# B&R Automation Studio project NAEUL004C00R13L518F00 (part 70)

#### Local.var - Do Not Change!!!
```iecst
(*2019-04-16*)
(**)
(*Local Action, State & Status*)
VAR
	eStatus : eFBStatus := Idle;
	udiStatus : UDINT := 0;
END_VAR
(**)
(*Local Alarm*)
VAR
	tyAlmData : tyAlmDat;
	a_tyAlmText : ARRAY[10000..10099] OF tyAlmTxt := [(sAlmText:='Magazine Not Present While Pushing Board Into Magazine',sRcyText:='Insert Magazine To Continue Operation.'),(sAlmText:='Conveyor Outlet Sensor Timeout Alarm',sRcyText:='Check Conveyor Outlet Sensor'),(sAlmText:='Conveyor Inlet Sensor Timeout Alarm',sRcyText:='Check Conveyor Inlet Sensor'),(sAlmText:='Clear Sensor Activated When Board Transfer In',sRcyText:='Please Check The Sensitivity of Pusher Conveyor Outlet Sensor'),(sAlmText:='Magazine Width Check Timeout Alarm',sRcyText:='Magazine Is Not Set In Correct Width'),(sAlmText:='Pusher AntiJam Sensor On',sRcyText:='Board Jam During Pusher Is Extending'),(sAlmText:='No Barcode Detected.',sRcyText:='Check The Barcode Position.'),(sAlmText:='Return Code Feedback Time Out.',sRcyText:='Reset And Resume Operation.'),(sAlmText:='Board Lost Before Traversing.',sRcyText:='Check If Outlet sensor False Triggerred or Board Stuck in Middle '),(sAlmText:='Inlet and outlet same time sensing error.',sRcyText:='Please Ensure No Blockage At Inlet Sensor.'),(sAlmText:='OpCon Error',sRcyText:='OpCon Error'),(sAlmText:='ScanningTime Out Error',sRcyText:='Ensure Connection for Scan Completed Signal'),(sAlmText:='Anti Crash Sensor Activated Before Traversing',sRcyText:='Please Check Board is away from Clear Sensor'),87((0))];
END_VAR
(**)
(*Local Output*)
VAR
	sStepTxt : STRING[80];
	bPaused : BOOL;
END_VAR
(**)
VAR
	eUSSMEMAAct1 : eSMEMAAction;
	eUSSMEMAAct2 : eSMEMAAction;
	eUSSMEMAAct3 : eSMEMAAction;
	eDSSMEMAAct1 : eSMEMAAction;
	eDSSMEMAAct2 : eSMEMAAction;
	eDSSMEMAAct3 : eSMEMAAction;
	eConvAct : eConvAction;
	eAWAct : eAWAction;
	eAWPushOrPullerAct : eAWAction;
	eTravAct : eTravAction;
	eLifAct : eLifterAction;
	eInletPneuAct : ePneuAction;
	eOutletPneuAct : ePneuAction;
	eOutletPneuAct2 : ePneuAction;
	eOutletPneuAct3 : ePneuAction;
	eStopperAct1 : ePneuAction;
	eStopperAct2 : ePneuAction;
	eStopperAct3 : ePneuAction;
	udiJogSpeed : UDINT := 290000;
END_VAR
(**)
VAR
	eTravLifPosGo : eTravLifULPos;
	a_bMagDis : ARRAY[1..3] OF BOOL;
	a_bMagRej : ARRAY[1..3] OF BOOL;
	bInitConv : BOOL;
	bOpsInitDone : BOOL;
	bUSComm : BOOL;
	bEntBrd : BOOL;
	bDSComm : BOOL;
	bExitBrd : BOOL;
	bTravLifMove : BOOL;
	bUSWidthChkBrdExist : BOOL := TRUE;
	bStopperExtStep : BOOL;
	fbWaitTimer : TON := (PT:=T#2s);
	fbWidthChkSenOnTim : TON := (PT:=T#5s);
	fbWidthChkSenOffTim : TON := (PT:=T#1s);
END_VAR
(*Step Logger*)
VAR
	bClsLog : BOOL;
	blog : BOOL;
	logStep : ARRAY[0..999] OF eTravLifULStep;
	logIndexStep : INT;
	eGotoOpsStepDummy : eTravLifULStep;
END_VAR
(**)
(*Local Input*)
VAR
	udiRstErr : UDINT := 0;
	bEn : BOOL := TRUE;
	bDis : BOOL := FALSE;
	bRun : BOOL;
	bStop : BOOL;
	bStep : BOOL;
	eULMode : eULMod;
	eULMagazine : eULMag;
	bNonBffrMod : BOOL;
	bBypsGdBadBrd : BOOL;
	bUSAllow : BOOL := TRUE;
	bDSAllow : BOOL := TRUE;
	eUSCommMod1 : eMcSetCommMod;
	eUSCommMod2 : eMcSetCommMod;
	eUSCommMod3 : eMcSetCommMod;
	eDSCommMod1 : eMcSetCommMod;
	eDSCommMod2 : eMcSetCommMod;
	eDSCommMod3 : eMcSetCommMod;
	eUSSMEMAStat1 : eSMEMAAction;
	eUSSMEMAStatus1 : eFBStatus;
	bUSSMEMAUSRdy1 : BOOL;
	bUSSMEMAGdBrdRdy1 : BOOL;
	bUSSMEMATransporting1 : BOOL;
	bUSSMEMAConvStart1 : BOOL;
	bUSSMEMAConvStop1 : BOOL;
	eUSSMEMAStat2 : eSMEMAAction;
	eUSSMEMAStatus2 : eFBStatus;
	bUSSMEMAUSRdy2 : BOOL;
	bUSSMEMAGdBrdRdy2 : BOOL;
	bUSSMEMATransporting2 : BOOL;
	bUSSMEMAConvStart2 : BOOL;
	bUSSMEMAConvStop2 : BOOL;
	eUSSMEMAStat3 : eSMEMAAction;
	eUSSMEMAStatus3 : eFBStatus;
	bUSSMEMAUSRdy3 : BOOL;
	bUSSMEMAGdBrdRdy3 : BOOL;
	bUSSMEMATransporting3 : BOOL;
	bUSSMEMAConvStart3 : BOOL;
	bUSSMEMAConvStop3 : BOOL;
	eDSSMEMAStat1 : eSMEMAAction;
	eDSSMEMAStatus1 : eFBStatus;
	bDSSMEMADSRdy1 : BOOL;
	bDSSMEMAConvStart1 : BOOL;
	eDSSMEMAStat2 : eSMEMAAction;
	eDSSMEMAStatus2 : eFBStatus;
	bDSSMEMADSRdy2 : BOOL;
	bDSSMEMAConvStart2 : BOOL;
	eDSSMEMAStat3 : eSMEMAAction;
	eDSSMEMAStatus3 : eFBStatus;
	bDSSMEMADSRdy3 : BOOL;
	bDSSMEMAConvStart3 : BOOL;
	bUSHermesUSRdy1 : BOOL;
	bUSHermesUSGdRdy1 : BOOL;
	bUSHermesTransporting1 : BOOL;
	bUSHermesStopTransport1 : BOOL;
	bUSHermesUSRdy2 : BOOL;
	bUSHermesUSGdRdy2 : BOOL;
	bUSHermesTransporting2 : BOOL;
	bUSHermesStopTransport2 : BOOL;
	bUSHermesUSRdy3 : BOOL;
	bUSHermesUSGdRdy3 : BOOL;
	bUSHermesTransporting3 : BOOL;
	bUSHermesStopTransport3 : BOOL;
	bDSHermesDSRdy1 : BOOL;
	bDSHermesTransporting1 : BOOL;
	bDSHermesStopTransport1 : BOOL;
	bDSHermesDSRdy2 : BOOL;
	bDSHermesTransporting2 : BOOL;
	bDSHermesStopTransport2 : BOOL;
	bDSHermesDSRdy3 : BOOL;
	bDSHermesTransporting3 : BOOL;
	bDSHermesStopTransport3 : BOOL;
	eConvStat : eConvAction;
	eConvStatus : eFBStatus;
	eConvDirection : eConvDir;
	bConvHvBrd : BOOL;
	bConvGdBrd : BOOL;
	eAWStat : eAWAction;
	eAWStatus : eFBStatus;
	bAWWidthPosDiff : BOOL;
	eTravStat : eTravAction;
	eTravStatus : eFBStatus;
	eLifStat : eLifterAction;
	eLifStatus : eFBStatus;
	eInletPneuStat : ePneuAction;
	eInletPneuStatus : eFBStatus;
	bInletPneuCls : BOOL;
	eOutletPneuStat : ePneuAction;
	eOutletPneuStatus : eFBStatus;
	bConvLftSen : BOOL;
	bConvRgtSen : BOOL;
	bMagTransferBrd1 : BOOL;
	bMagTransferBrd2 : BOOL;
	bMagTransferBrd3 : BOOL;
	bBufferMagPresent1 : BOOL;
	bBufferMagPresent2 : BOOL;
	bBufferMagPresent3 : BOOL;
	sProgNm : STRING[15] := 'Ops TravLifUL';
	bNtSettingsLoadDone : BOOL := TRUE;
	tShutterWaitTmr : TIME := T#0s;
	eMagBuffferActLoad : eLifMagULUpdateData;
	bScanEn : BOOL := FALSE;
	eTCPTopStat : eTCPAction1;
	eTCPTopStatus : eFBStatus;
	sTopMsgRd : STRING[80] := '';
	eTCPBtmStat : eTCPAction1;
	eTCPBtmStatus : eFBStatus;
	sBtmMsgRd : STRING[80] := '';
	bInitInletPneu : BOOL := FALSE;
	bWidthChkErrCmdUnclmp1 : BOOL;
	bWidthChkErrCmdUnclmp2 : BOOL;
	bWidthChkErrCmdUnclmp3 : BOOL;
	bCmdUnclmpFlag : BOOL;
	bPneuUnclmpFBDone : BOOL;
END_VAR
(**)
(*Local*)
VAR
	bRstErr : BOOL;
	udiRstErrOld : UDINT;
	bInitDone : BOOL;
	bInitialDone : BOOL;
	eOpsStep : eTravLifULStep := TravLifULStepNA;
	eGotoOpsStep : eTravLifULStep := TravLifULStepInitConv;
	tyParamTravLif : tyParamTravLifUL;
	bOpsModGonethrough : BOOL;
	udiMagPresentTm1 : UDINT;
	udiMagPresentTm : UDINT;
	udiCmpTm : UDINT;
	udiCount : UDINT;
	udi : UDINT;
	bGdChk : BOOL;
	udiPosAllwGo : UDINT;
	a_bPosAllwSigOn : ARRAY[1..3] OF BOOL;
	a_udiPosAllwSum : ARRAY[1..3] OF UDINT;
	a_tyMagAllwBffrStat : ARRAY[1..3] OF tyBffrStat;
	a_udiMagAllwMagPresentTm : ARRAY[1..3] OF UDINT;
	a_udiMagAllwPriority : ARRAY[1..3] OF UDINT;
	bBrdOnSen : BOOL;
	bBrdOnStopperSen : BOOL;
	bStopperBrdOnSen : BOOL;
	bConvInSenOn : BOOL;
	bConvOutSenOn : BOOL;
	bLocalUSRdy1 : BOOL;
	bLocalUSGdRdy1 : BOOL;
	bLocalUSRdy2 : BOOL;
	bLocalUSGdRdy2 : BOOL;
	bLocalUSRdy3 : BOOL;
	bLocalUSGdRdy3 : BOOL;
	bLocalDSRdy1 : BOOL;
	bLocalDSRdy2 : BOOL;
	bLocalDSRdy3 : BOOL;
	bSkipCloseInletShutter : BOOL;
	tConvRgtSenOff : TON := (PT:=T#100ms);
	tConvLftSenOff : TON := (PT:=T#100ms);
	tEntBoardTimoutErr : TON := (PT:=T#6s);
	tExitBoardTimoutErr : TON := (PT:=T#10s);
	tTravLiftInPos : TON := (PT:=T#100ms);
	bTravLifInDSPos : BOOL;
	bSelfTest : BOOL;
	bLifterBtmPosDiff : BOOL;
	bLifterAPosDiff : BOOL;
	bLifterBPosDiff : BOOL;
	bBypCurtainSenPB : BOOL;
	bBypCurtainSenCtrl : BOOL;
	bBypCurtainSensorPBLED : BOOL;
	bMagWidthChkDis : BOOL;
	fbRstCurtain : TON := (PT:=T#1m);
	fb2SenTm : TON;
	p_eStopperAct : REFERENCE TO ePneuAction;
	p_eStopperStat : REFERENCE TO ePneuAction;
	p_eStopperStatus : REFERENCE TO eFBStatus;
	p_bStopperBlk : REFERENCE TO BOOL;
	p_eLocalUSCommMod : REFERENCE TO eMcSetCommMod;
	p_eLocalDSCommMod : REFERENCE TO eMcSetCommMod;
	p_bLocalUSRdy : REFERENCE TO BOOL;
	p_bLocalUSGdRdy : REFERENCE TO BOOL;
	p_bLocalDSRdy : REFERENCE TO BOOL;
	p_eLocalUSSMEMAAct : REFERENCE TO eSMEMAAction;
	p_eLocalUSSMEMAStat : REFERENCE TO eSMEMAAction;
	p_eLocalUSSMEMAStatus : REFERENCE TO eFBStatus;
	p_bLocalUSSMEMAUSRdy : REFERENCE TO BOOL;
	p_bLocalUSSMEMAGdBrdRdy : REFERENCE TO BOOL;
	p_bLocalUSSMEMATransporting : REFERENCE TO BOOL;
	p_bLocalUSSMEMAConvStart : REFERENCE TO BOOL;
	p_bLocalUSSMEMAConvStop : REFERENCE TO BOOL;
	p_eLocalDSSMEMAAct : REFERENCE TO eSMEMAAction;
	p_eLocalDSSMEMAStat : REFERENCE TO eSMEMAAction;
	p_eLocalDSSMEMAStatus : REFERENCE TO eFBStatus;
	p_bLocalDSSMEMADSRdy : REFERENCE TO BOOL;
	p_bLocalDSSMEMAConvStart : REFERENCE TO BOOL;
	p_bLocalUSHermesUSRdy : REFERENCE TO BOOL;
	p_bLocalUSHermesUSGdRdy : REFERENCE TO BOOL;
	p_bLocalUSHermesTransporting : REFERENCE TO BOOL;
	p_bLocalUSHermesStopTransport : REFERENCE TO BOOL;
	p_bLocalDSHermesDSRdy : REFERENCE TO BOOL;
	p_bLocalDSHermesTransporting : REFERENCE TO BOOL;
	p_bLocalDSHermesStopTransport : REFERENCE TO BOOL;
	fbBypCurtainPBLEDBlinkTm : TON := (IN:=FALSE,PT:=T#500ms,Q:=FALSE,ET:=0,StartTime:=0,M:=FALSE,Restart:=0);
	eLocalUSCommMod : eMcSetCommMod;
	bWait : BOOL;
END_VAR
(*Inlet stopper*)
VAR
	eInletStopperAct : ePneuAction;
END_VAR
(*Scanner Param *)
VAR
	eTCPTopAct : eTCPAction1;
	eTCPBtmAct : eTCPAction1;
	sBarcode : STRING[80];
	bPass : BOOL;
END_VAR
(*xml*)
VAR
	tyOpConParam : tyLocationParam;
	tyOpConMsgReq : eOpConMsgType;
	bJamStarted : BOOL := FALSE;
	bWaitMagChkRetCode : BOOL;
	fbIdleTm : TON := (PT:=T#3m);
	fbReturnCodeTO : TON := (PT:=T#30s);
END_VAR
(**)
VAR
	tyPartReceive : tyOpConPartReceive;
	tyPartProcessedItems : tyOpConPartProcessed; (*Output*)
	tyMagCoordinate : tyMagCoord;
	diTemp : DINT;
	bHermesBC : BOOL;
	diMagBrdQty : ARRAY[1..3] OF DINT;
	bPLCGrabPic : BOOL;
	asMagEntered : ARRAY[0..4] OF STRING[10];
	udiModuleNum : UDINT := 6621;
END_VAR
(*Siemen *)
VAR
	bAllwExitMag1 : BOOL;
	bAllwExitMag2 : BOOL;
	bAllwExitMag3 : BOOL;
	fbInletStopperOffTim : TON := (PT:=T#1s);
END_VAR
(*Bosch Scanner*)
VAR
	bScannerEn : BOOL;
	bTCPScanner : BOOL;
	bSignalTrigMagOutEn : BOOL;
	bTCPScannerEn : BOOL;
	fbScanTimOut : TON := (PT:=T#10s);
	bStartScanSig : BOOL;
	bPCBExitMag1 : BOOL;
	bPCBExitMag2 : BOOL;
	bPCBExitMag3 : BOOL;
	usiScanCntr : USINT;
END_VAR
```

### OpsMagConvUL.typ - Do Not Change!!!
```iecst
(*2018-12-11*)
(**)
(*Sequence*)

TYPE
	eMagConvULStep :
		(
		MagConvULStepNA,
		MagConvULStepInitMag,
		MagConvULStepSafetyBarExtCtrl,
		MagConvULStepMagUSComm,
		MagConvULStepInitAWPneu,
		MagConvULStepInitMagEnt,
		MagConvULStepInitMagFixClp,
		MagConvULStepInitMagConv,
		MagConvULStepMagEnt,
		MagConvULStepMagEntMnl,
		MagConvULStepSelClampCtrl,
		MagConvULStepVerifyMag,
		MagConvULStepChkMag,
		MagConvULStepSafetyBarExt,
		MagConvULStepSafetyBarRet,
		MagConvULStepMagAWEngage,
		MagConvULStepMagAWDisengage,
		MagConvULStepMagAWHm,
		MagConvULStepMagAWMov,
		MagConvULStepMagEntMESStdByChk,
		MagConvULStepBffrStatChk,
		MagConvULStepMagCmp,
		MagConvULStepMtyBffr,
		MagConvULStepNxtLoadBffr,
		MagConvULStepBffrUSComm,
		MagConvULStepBffrEntBrd,
		MagConvULStepUpdateBffr,
		MagConvULStepLoadBffr,
		MagConvULStepMagExtMESStdByChk,
		MagConvULStepMagExitClampCtrl,
		MagConvULStepMagExitSafeBarCtrl,
		MagConvULStepMagFullDSComm,
		MagConvULStepMagFullExit,
		MagConvULStepMagExitMnl,
		MagConvULStepMagHalfExitMnl,
		MagConvULStepMagExitedWait,
		MagConvULStepMagExitedAGVWait
		);
	eLifMagULUpdateData :
		(
		BufferActLoadWhenStarted,
		BufferActLoadWhenCompleted
		);
END_TYPE
```

### OpsMagConvUL1.var - Change By Project
```iecst
(*2019-03-25*)
(**)
(*Action & State & Status*)
(**)
(*Alarm*)
VAR
	p_OpsMagConvUL1AlmData : UDINT;
	p_OpsMagConvUL1AlmData1 : UDINT;
END_VAR
(**)
(*Output*)
VAR
	p_OpsMagConvUL1StepTxt : UDINT;
	p_OpsMagConvUL1Paused : UDINT;
END_VAR
(**)
VAR
	p_OpsMagConvUL1BufferAct : UDINT;
	p_OpsMagConvUL1MagConv2ClpAct : UDINT;
	p_OpsMagConvUL1USSMEMAAct : UDINT;
	p_OpsMagConvUL1AGVMagAct : UDINT;
	p_OpsMagConvUL1MagFullExit : UDINT;
	p_OpsMagConvUL1IncorrectMagModel : UDINT;
	p_OpsMagConvUL1MagSizeL : UDINT;
END_VAR
(**)
VAR
	p_OpsMagConvUL1InitDone : UDINT;
	p_OpsMagConvUL1MagBffrAvl : UDINT;
	p_OpsMagConvUL1NewMagAllw : UDINT;
	p_OpsMagConvUL1RlsMagAllw : UDINT;
	p_OpsMagConvUL1EjectMESStep : UDINT;
	p_OpsMagConvUL1EjectMagNotAllw : UDINT;
	p_OpsMagConvUL1StepSelClampCtrl : UDINT;
	p_OpsMagConvUL1StepMagExitedWait : UDINT;
	p_OpsMagConvUL1NewMagVerified : UDINT;
	p_OpsMagConvUL1StepUSCom : UDINT;
	p_OpsMagConvUL1StepBffrLoad : UDINT;
	p_OpsMagConvUL1StepPLCGrab : UDINT;
END_VAR
(**)
VAR
	p_OpsMagConvUL1SafetyBarAct : UDINT;
	p_OpsMagConvUL1MagAWEngageAct : UDINT;
	p_OpsMagConvUL1MagAWAct : UDINT;
	p_OpsAGVCommRdy1 : UDINT;
END_VAR
(**)
VAR
	p_OpsMagConvUL1USSOTAct : UDINT;
	p_OpsMagConvUL1DSSOTAct : UDINT;
	p_OpsMagConvUL1MsgReq : UDINT;
	p_OpsMagConvUL1UnclmpDone : UDINT;
	p_OpsMagConvUL1MagAllwGo : UDINT;
	p_OpsMagConvUL1ReadRFID : UDINT;
	p_OpsMagConvUL1WriteRFID : UDINT;
	p_OpsMagConvUL1AWDone : UDINT;
	p_OpsMagConvUL1SlotUpdtDone : UDINT;
	p_OpsMagConvUL1AcptTm : UDINT;
	p_OpsMagConvUL1MESAcptCond : UDINT;
	p_OpsMagConvUL1MagExitedWait : UDINT;
	p_OpsMagConvUL1TLMuteBuzz : UDINT;
	p_OpsMagConvUL1MagFullInfo : UDINT;
END_VAR
(**)
```

### Program Logical/Operations/MagConv_StationaryPlat/OpsMagConvUL1 (IEC) - 1.00.0 - 

#### InputRef.var
```iecst
(*2019-04-16*)
(**)
(*General*)
VAR
	p_udiRstErr : REFERENCE TO UDINT;
	p_bEn : REFERENCE TO BOOL;
	p_bDis : REFERENCE TO BOOL;
	p_bRun : REFERENCE TO BOOL;
	p_bStop : REFERENCE TO BOOL;
	p_bStep : REFERENCE TO BOOL;
END_VAR
(**)
(*Configuration*)
VAR
	p_sProgNm : REFERENCE TO STRING[15];
	p_bNtSettingsLoadDone : REFERENCE TO BOOL;
END_VAR
(**)
VAR
	p_usiMagConv : REFERENCE TO USINT;
	p_bInfoEn : REFERENCE TO BOOL;
END_VAR
(**)
VAR
	pa_bMagDis : REFERENCE TO ARRAY[1..3] OF BOOL;
	pa_bMagRej : REFERENCE TO ARRAY[1..3] OF BOOL;
	pa_bMagChangeOverBlk : REFERENCE TO ARRAY[1..4] OF BOOL;
	p_bMagPropDiffBlk : REFERENCE TO BOOL;
	p_bUSAllow : REFERENCE TO BOOL;
	p_bAllwChgWidth : REFERENCE TO BOOL;
	p_bAllwChgSlot : REFERENCE TO BOOL;
	p_bChgMagWidth : REFERENCE TO BOOL;
	p_bChgMagSlot : REFERENCE TO BOOL;
	p_bMagOrientChkSenPrep : REFERENCE TO BOOL;
	p_bDIMagFixedClampSen : REFERENCE TO BOOL;
	p_eCustomerReq : REFERENCE TO eCustomer;
END_VAR
(*Siemen MES*)
VAR
	p_tyResponseFromMES : REFERENCE TO tyStatPlatformFromMES;
	p_bOpsTravLifAllwExitMag : REFERENCE TO BOOL;
	p_diMcParamMESResponseTO : REFERENCE TO DINT;
	p_bMcParamMESEn : REFERENCE TO BOOL;
	p_bAutoRcpForceExitMag : REFERENCE TO BOOL;
	p_dtCurrDT : REFERENCE TO DATE_AND_TIME;
	p_dtOpsMagConvUL1AcptTm : REFERENCE TO DATE_AND_TIME;
	p_dtOpsMagConvUL2AcptTm : REFERENCE TO DATE_AND_TIME;
	p_dtOpsMagConvUL3AcptTm : REFERENCE TO DATE_AND_TIME;
	p_iOpsMagConvUL1MESAcptCond : REFERENCE TO INT;
	p_iOpsMagConvUL2MESAcptCond : REFERENCE TO INT;
	p_iOpsMagConvUL3MESAcptCond : REFERENCE TO INT;
	p_bOpsMagConvUL2MagExitedWait : REFERENCE TO BOOL;
	p_bOpsMagConvUL3MagExitedWait : REFERENCE TO BOOL;
	p_usiUIHcomModchanged : REFERENCE TO USINT;
	p_bNtParamAutoRcpF1ArbitraryType : REFERENCE TO BOOL;
END_VAR
(**)
VAR
	p_bNewMag : REFERENCE TO BOOL;
	p_bRlsMag : REFERENCE TO BOOL;
END_VAR
(**)
VAR
	p_bConvInitDone : REFERENCE TO BOOL;
	p_bConvHvBrd : REFERENCE TO BOOL;
	p_bConvGdBrd : REFERENCE TO BOOL;
END_VAR
(**)
VAR
	p_tyBufferStat1 : REFERENCE TO tyBffrStat;
	p_tyBufferStat2 : REFERENCE TO tyBffrStat;
	p_tyBufferStat3 : REFERENCE TO tyBffrStat;
END_VAR
(**)
VAR
	p_bMagClampRS1 : REFERENCE TO BOOL;
	p_bMagClampRS2 : REFERENCE TO BOOL;
	p_bMagClampRS3 : REFERENCE TO BOOL;
END_VAR
(**)
VAR
	p_bMagEntrySen : REFERENCE TO BOOL;
	p_bMagEntrySen1 : REFERENCE TO BOOL;
	p_bMagEntrySen2 : REFERENCE TO BOOL;
	p_bMagEntrySen3 : REFERENCE TO BOOL;
END_VAR
(**)
VAR
	p_bMagPresentSen : REFERENCE TO BOOL;
	p_bMagPresentSen1 : REFERENCE TO BOOL;
	p_bMagPresentSen2 : REFERENCE TO BOOL;
	p_bMagPresentSen3 : REFERENCE TO BOOL;
END_VAR
(**)
VAR
	p_bBufferMagPresent1 : REFERENCE TO BOOL;
	p_bBufferMagPresent2 : REFERENCE TO BOOL;
	p_bBufferMagPresent3 : REFERENCE TO BOOL;
END_VAR
(**)
VAR
	p_bBufferMagRemoved : REFERENCE TO BOOL;
	p_bBufferMagRemoved1 : REFERENCE TO BOOL;
	p_bBufferMagRemoved2 : REFERENCE TO BOOL;
	p_bBufferMagRemoved3 : REFERENCE TO BOOL;
END_VAR
(**)
VAR
	p_dtBufferMagPresentTm1 : REFERENCE TO DATE_AND_TIME;
	p_dtBufferMagPresentTm2 : REFERENCE TO DATE_AND_TIME;
	p_dtBufferMagPresentTm3 : REFERENCE TO DATE_AND_TIME;
END_VAR
(**)
VAR
	p_eBufferStat : REFERENCE TO eBufferAction;
	p_eBufferStatus : REFERENCE TO eFBStatus;
END_VAR
(**)
VAR
	p_eMagConv2ClpStat : REFERENCE TO eMagConv2ClpAction;
	p_eMagConv2ClpStatus : REFERENCE TO eFBStatus;
	p_bMagConv2ClpHvMag : REFERENCE TO BOOL;
END_VAR
(**)
VAR
	p_eUSSMEMAStat : REFERENCE TO eSMEMAAction;
	p_eUSSMEMAStatus : REFERENCE TO eFBStatus;
	p_bUSSMEMATransporting : REFERENCE TO BOOL;
	p_bUSSMEMAConvStart : REFERENCE TO BOOL;
	p_bUSSMEMAConvStop : REFERENCE TO BOOL;
END_VAR
(**)
VAR
	p_eAGVMagStat : REFERENCE TO eAGVMagAction;
	p_eAGVMagStatus : REFERENCE TO eFBStatus;
	p_bAGVMagMcRunRdy : REFERENCE TO BOOL;
	p_tyAGVToDTMag : REFERENCE TO tyTagAGVToDTMag;
END_VAR
(**)
VAR
	p_eSelClampCtrlStat : REFERENCE TO ePneuAction;
	p_eSelClampCtrlStatus : REFERENCE TO eFBStatus;
END_VAR
(**)
VAR
	p_bOutShutterExtended : REFERENCE TO BOOL;
END_VAR
(**)
VAR
	p_bDIMagConvHeightSen : REFERENCE TO BOOL;
	p_bDIMagConvSelUnclampRS : REFERENCE TO BOOL;
	p_bDIMagConvCAB717Sen : REFERENCE TO BOOL;
	p_bDIMagConvSmallSen : REFERENCE TO BOOL;
	p_bDIMagConvLargeSen : REFERENCE TO BOOL;
	p_bDIOutShutterClosedRS : REFERENCE TO BOOL;
END_VAR
(**)
VAR
	p_eSafetyBarStat : REFERENCE TO ePneuAction;
	p_eSafetyBarStatus : REFERENCE TO eFBStatus;
	p_bSafetyBarExtended : REFERENCE TO BOOL;
	p_bSafetyBarRetracted : REFERENCE TO BOOL;
END_VAR
(**)
VAR
	p_eMagAWEngageStat : REFERENCE TO ePneuAction;
	p_eMagAWEngageStatus : REFERENCE TO eFBStatus;
	p_eConvStat : REFERENCE TO eConvAction;
	p_eConvStatus : REFERENCE TO eFBStatus;
END_VAR
(**)
VAR
	p_eMagAWStat : REFERENCE TO eMagAWAction;
	p_eMagAWStatus : REFERENCE TO eFBStatus;
	p_bMagAWEngaging : REFERENCE TO BOOL;
	p_bMagAWErr : REFERENCE TO BOOL;
	p_bMagAWOpenLimit : REFERENCE TO BOOL;
	p_bMagAWCloseLimit : REFERENCE TO BOOL;
END_VAR
(**)
VAR
	p_eUSSOTStat : REFERENCE TO eSOTAction;
	p_eUSSOTStatus : REFERENCE TO eFBStatus;
	p_bUSSOTTransporting : REFERENCE TO BOOL;
	p_bUSSOTConvStart : REFERENCE TO BOOL;
	p_bUSSOTConvStop : REFERENCE TO BOOL;
	p_bUSSOTUSRdy : REFERENCE TO BOOL;
	p_bUSSOTUSLargeMagRdy : REFERENCE TO BOOL;
END_VAR
(**)
VAR
	p_eDSSOTStat : REFERENCE TO eSOTAction;
	p_eDSSOTStatus : REFERENCE TO eFBStatus;
	p_bDSSOTConvStart : REFERENCE TO BOOL;
	p_bDSSOTConvStop : REFERENCE TO BOOL;
END_VAR
(**)
VAR
	p_bOpsTravLifExitBrd : REFERENCE TO BOOL;
	p_bOpsTravLifMov : REFERENCE TO BOOL;
END_VAR
(**)
(*Self Test Var*)
VAR
	p_bSelfTest : REFERENCE TO BOOL;
	p_bMcParamMagAWDis : REFERENCE TO BOOL;
	p_bDISOTRcv : REFERENCE TO BOOL;
	p_bDISOTAGVReady : REFERENCE TO BOOL;
END_VAR
(**)
VAR
	p_diProdRcpCurrRcp1Width : REFERENCE TO DINT;
	p_diProdRcpCurrRcp2Width : REFERENCE TO DINT;
	p_sProdRcpCurrRcp1Name : REFERENCE TO STRING[80];
	p_sProdRcpCurrRcp2Name : REFERENCE TO STRING[80];
	p_sMagRcpName : REFERENCE TO DINT;
	p_bOpsTravLifErrCmdUnclmp : REFERENCE TO BOOL;
END_VAR
(**)
VAR
	p_bNtParamAutoRcpPrep : REFERENCE TO BOOL;
	p_bMcParamAutoRcpDis : REFERENCE TO BOOL;
END_VAR
```

#### InputRef_Link.var
```iecst
(*2018-12-11*)
(**)
VAR
	p_bLinkDIMagPresentSen1 : REFERENCE TO BOOL;
	p_bLinkMagConv2Clp1MtrIn : REFERENCE TO BOOL;
	p_bLinkMagConv2Clp1MtrOut : REFERENCE TO BOOL;
	p_bLinkDIMagPresentSen2 : REFERENCE TO BOOL;
	p_bLinkMagConv2Clp2MtrIn : REFERENCE TO BOOL;
	p_bLinkMagConv2Clp2MtrOut : REFERENCE TO BOOL;
	p_bLinkDIMagPresentSen3 : REFERENCE TO BOOL;
	p_bLinkMagConv2Clp3MtrIn : REFERENCE TO BOOL;
	p_bLinkMagConv2Clp3MtrOut : REFERENCE TO BOOL;
	p_bLinkFixedMagClampRS1 : REFERENCE TO BOOL;
	p_bLinkRmtMagClampRS1 : REFERENCE TO BOOL;
	p_bLinkFixedMagClampRS2 : REFERENCE TO BOOL;
	p_bLinkRmtMagClampRS2 : REFERENCE TO BOOL;
	p_bLinkFixedMagClampRS3 : REFERENCE TO BOOL;
	p_bLinkRmtMagClampRS3 : REFERENCE TO BOOL;
	p_bLinkMcParamMagAutoDetTm : REFERENCE TO DINT;
	p_bLinkDIMagEntrySen : REFERENCE TO BOOL;
	p_bLinkNtParamMagModelAutoVerify : REFERENCE TO BOOL;
	p_bLinkMagRcpCurrRcpMagModel : REFERENCE TO USINT;
	p_bLinkNewMagVerified2 : REFERENCE TO BOOL;
	p_bLinkNewMagVerified3 : REFERENCE TO BOOL;
	p_eNtParamProjMagBuffferActLoad : REFERENCE TO eLifMagULUpdateData;
	p_eLinkMcParamMagExMode : REFERENCE TO eMcMagExchangeMode;
END_VAR
(**)
VAR
	p_bMag1OrientationChkSen1 : REFERENCE TO BOOL;
	p_bMagHeightDetSen1 : REFERENCE TO BOOL;
	p_bMagHeightDetEn : REFERENCE TO BOOL;
	p_bMagHeightDetPrep : REFERENCE TO BOOL;
	p_bProjLifTravMnlLoad : REFERENCE TO BOOL;
END_VAR
```

#### Local.var
```iecst
(*2019-04-16*)
(**)
(*Local Action, State & Status*)
VAR
	eStatus : eFBStatus := Idle;
	udiStatus : UDINT := 0;
	udiStatus1 : UDINT := 0;
END_VAR
(**)
(*Local Alarm*)
VAR
	tyAlmData : tyAlmDat;
	tyAlmData1 : tyAlmDat;
	a_tyAlmText : ARRAY[10000..10099] OF tyAlmTxt := [(sAlmText:='Magazine Not Present'),(sAlmText:='Magazine 1 Is Full'),(sAlmText:='Magazine 2 Is Full'),(sAlmText:='Magazine 3 Is Full'),(sAlmText:='Please Insert Good Magazine'),(sAlmText:='Please Insert Bad Magazine'),(sAlmText:='Wrong Magazine Width On Position 1'),(sAlmText:='Wrong Magazine Height On Position 1'),(sAlmText:='Waiting for Unload Magazine 1'),(sAlmText:='Rack/Magazine Auto Width Change Error',sRcyText:='Rack/Magazine Auto Width Motor Error While Doing Width Change'),(sAlmText:='Magazine 1 Auto Width Limit Sensor Activated, Ensure Senor Is Cleared Or Magazine Is Empty ',sRcyText:='Please make sure magazine wall is clear from limit sensor and there is no object in the magazine'),(sAlmText:='Wrong Magazine Orientation Placed Or Wrong Magazine Loaded',sRcyText:='Please Check And Correct the Magazine Orientation/Reload Correct Magazine.'),(sAlmText:='Reading Mag 1 in Progress'),(sAlmText:='Reading Mag 1 or Press Release Mag'),(sAlmText:='Writing Mag 1'),(sAlmText:='Writing Mag 1 or Press Release Mag'),(sAlmText:='Wrong Magazine Position 1'),83(0)];
END_VAR
(**)
(*Local Output*)
VAR
	sStepTxt : STRING[80];
	bPaused : BOOL;
END_VAR
(**)
VAR
	eBufferAct : eBufferAction;
	eSelClampCtrl : ePneuAction;
	eMagConv2ClpAct : eMagConv2ClpAction;
	eUSSMEMAAct : eSMEMAAction;
	eAGVMagAct : eAGVMagAction;
END_VAR
(**)
VAR
	eSafetyBarAct : ePneuAction;
	eMagAWEngageAct : ePneuAction;
	eMagAWAct : eMagAWAction;
END_VAR
(**)
VAR
	eUSSOTAct : eSOTAction;
	eDSSOTAct : eSOTAction;
	bOpsInitDone : BOOL;
	bMagBffrAvl : BOOL;
	bNewMagAllw : BOOL;
	bRlsMagAllw : BOOL;
	bEjectMESStep : BOOL;
	bEjectMagNotAllw : BOOL;
	bStepMagExitedWait : BOOL;
	bStepMagVerification : BOOL;
	bStepMagFullExit : BOOL;
	bStepMagUSCom : BOOL;
	bStepMagBffrLoad : BOOL;
	bStepPLCGrab : BOOL;
END_VAR
(*Step Logger*)
VAR
	bClsLog : BOOL;
	blog : BOOL;
	logStep : ARRAY[0..999] OF eMagConvULStep;
	logIndexStep : INT;
	eGotoOpsStepDummy : eMagConvULStep;
END_VAR
(**)
(*Local Input*)
VAR
	udiRstErr : UDINT := 0;
	bEn : BOOL := TRUE;
	bDis : BOOL := FALSE;
	bRun : BOOL;
	bStop : BOOL;
	bStep : BOOL;
	usiMagConv : USINT;
	bInfoEn : BOOL := TRUE;
	a_bMagDis : ARRAY[1..3] OF BOOL;
	a_bMagRej : ARRAY[1..3] OF BOOL;
	bUSAllow : BOOL := TRUE;
	bAllwChgWidth : BOOL;
	bAllwChgSlot : BOOL;
	bNewMag : BOOL;
	bRlsMag : BOOL;
	bConvInitDone : BOOL;
	bConvHvBrd : BOOL;
	bConvGdBrd : BOOL;
	tyBufferStat1 : tyBffrStat;
	tyBufferStat2 : tyBffrStat;
	tyBufferStat3 : tyBffrStat;
	bMagClampRS1 : BOOL;
	bMagClampRS2 : BOOL;
	bMagClampRS3 : BOOL;
	bMagEntrySen1 : BOOL;
	bMagEntrySen2 : BOOL;
	bMagEntrySen3 : BOOL;
	bMagPresentSen1 : BOOL;
	bMagPresentSen2 : BOOL;
	bMagPresentSen3 : BOOL;
	bBufferMagPresent1 : BOOL;
	bBufferMagPresent2 : BOOL;
	bBufferMagPresent3 : BOOL;
	dtBufferMagPresentTm1 : DATE_AND_TIME;
	dtBufferMagPresentTm2 : DATE_AND_TIME;
	dtBufferMagPresentTm3 : DATE_AND_TIME;
	eBufferStat : eBufferAction;
	eBufferStatus : eFBStatus;
	eMagConv2ClpStat : eMagConv2ClpAction;
	eMagConv2ClpStatus : eFBStatus;
	bMagConv2ClpHvMag : BOOL;
	eUSSMEMAStat : eSMEMAAction;
	eUSSMEMAStatus : eFBStatus;
	bUSSMEMATransporting : BOOL;
	bUSSMEMAConvStart : BOOL;
	bUSSMEMAConvStop : BOOL;
	eAGVMagStat : eAGVMagAction;
	eAGVMagStatus : eFBStatus;
	bAGVMagMcRunRdy : BOOL;
	tyAGVToDualMag : tyTagAGVToDTMag;
	sProgNm : STRING[15] := 'Ops MagConvUL';
	bNtSettingsLoadDone : BOOL := TRUE;
END_VAR
(**)
(*Local*)
VAR
	bRstErr : BOOL;
	udiRstErrOld : UDINT;
	bInitDone : BOOL;
	bInitialDone : BOOL;
END_VAR
VAR RETAIN
	iMagMESAcptCond : INT;
	bMagExitedWait : BOOL;
	ePrevExitStep : eMagConvULStep;
END_VAR
VAR
	eOpsStep : eMagConvULStep := MagConvULStepNA;
	eGotoOpsStep : eMagConvULStep := MagConvULStepInitMag;
	udi : UDINT;
	udi1 : UDINT;
	udi2 : UDINT;
	udiCount : UDINT;
	udiCmpTm : UDINT;
	udiMagAllwGo : UDINT;
	a_tyMagAllwBffrStat : ARRAY[1..3] OF tyBffrStat;
	a_bMagAllwMagClamped : ARRAY[1..3] OF BOOL;
	a_bMagAllwMagPresent : ARRAY[1..3] OF BOOL;
	a_udiMagAllwMagPresentTm : ARRAY[1..3] OF UDINT;
	a_udiMagAllwPriority : ARRAY[1..3] OF UDINT;
	a_udiMagAllwSum : ARRAY[1..3] OF UDINT;
	p_tyLocalBufferStat : REFERENCE TO tyBffrStat;
	p_bLocalMagEntrySen : REFERENCE TO BOOL;
	p_bLocalBufferMagPresent : REFERENCE TO BOOL;
	p_dtLocalBufferMagPresentTm : REFERENCE TO DATE_AND_TIME;
	bPneuUnclmpDone : BOOL;
	usiPrevHcomModchanged : USINT;
END_VAR
(**)
VAR
	fbWrongMagTm : TON := (PT:=T#5000ms);
	fbMagAutoDetTm : TON := (PT:=T#2000ms);
	fbMagRemovedTm : TON := (PT:=T#1000ms);
	fbVerifyWarningDelay : TON := (PT:=T#1000ms);
	fbEntSenOff : TON := (PT:=T#1000ms);
	bNewMagAutoDetected : BOOL;
	bNewMagVerified : BOOL;
	bNewMagVerifyStarted : BOOL;
	bIncorrectMagazineModel : BOOL;
	bMagAWDone : BOOL;
	bWrongWidth : BOOL;
	bWrongHeight : BOOL;
	bMagSizeLarge : BOOL;
	bLimitSenActivated : BOOL;
END_VAR
VAR RETAIN
	bManualUnloadMag : BOOL;
END_VAR
VAR
	bAIVInPos : BOOL;
	bCAB703 : BOOL;
	bFIXMag : BOOL;
	bMagManEx : BOOL;
	bMagAutoEx : BOOL;
	bAGVComm1Rdy : {REDUND_UNREPLICABLE} BOOL;
	bTLMuteBuzzer : BOOL;
	bMagFullInfo : BOOL;
	bStepOpsMagAWDone : BOOL;
	bStepOpsPitchUpdated : BOOL;
END_VAR
(*xml*)
VAR
	tyOpConParam : tyLocationParam;
	tyOpConMsgReq : eOpConMsgType;
	bPartMissingStarted : BOOL := FALSE;
	fbIdleTm : TON := (PT:=T#3m);
	udiModuleNum : UDINT := 6661;
END_VAR
(*ForSiemen*)
VAR
	bAutoRcpEn : BOOL;
	ePrevStepBeforeMESStdBy : eMagConvULStep;
	bWriteRFID : BOOL;
	bReadRFID : BOOL;
	fbReadRFIDTO : TON := (PT:=T#3s);
	fbWriteRFIDTO : TON;
END_VAR
VAR RETAIN
	dtMagConvAcptTm : DATE_AND_TIME;
END_VAR
VAR
	a_iMagMESAcptCond : ARRAY[1..3] OF INT;
END_VAR
```

#### Act_Alarm.st
```iecst
(** 2019-03-25 **)
ACTION Act_Alarm:

	//Error
	IF EDGEPOS(eStatus = Error) THEN

		tyAlmData.sProgNm		:= p_sProgNm;
		tyAlmData.udiCode		:= udiStatus;
		tyAlmData.eSeverity		:= AlmSeverityError;
		tyAlmData.udiRunTime	:= tyAlmData.udiRunTime + 1;
		tyAlmData.bAlm			:= TRUE;
		tyAlmData.udiModuleNum  := udiModuleNum;
		g_sOpsMagConvULProgNm		:= p_sProgNm;

		//Get Error Message
		IF tyAlmData.udiCode < 10000 OR tyAlmData.udiCode > 10099 THEN
			tyAlmData.sAlmMsg	:= 'Unknown';
			tyAlmData.sRcyMsg	:= 'Unknown';
		ELSE
			tyAlmData.sAlmMsg	:= a_tyAlmText[tyAlmData.udiCode].sAlmText;
			tyAlmData.sRcyMsg	:= a_tyAlmText[tyAlmData.udiCode].sRcyText;
		END_IF

	ELSIF bRstErr AND (tyAlmData.udiCode <> 0) THEN

		tyAlmData.udiCode		:= 0;
		tyAlmData.eSeverity		:= AlmSeverityNA;
		tyAlmData.sAlmMsg		:= '';
		tyAlmData.sRcyMsg		:= '';
		tyAlmData.bAlm			:= FALSE;
	END_IF

END_ACTION
```

#### Act_Background.st
```iecst
(** 2019-04-16 **)
ACTION Act_Background:

	//Reset bPaused
	IF EDGENEG(p_bStop OR p_bStep) THEN
		bPaused	:= FALSE;
	END_IF

	IF eStatus <> Error AND p_bRun = TRUE THEN
		IF (p_bEn = TRUE) AND (p_bDis = FALSE) THEN
			Act_OpsRun;
		ELSE
			bPaused	:= p_bStop OR p_bStep;
		END_IF

		IF EDGEPOS(p_bEn = FALSE OR p_bDis = TRUE) THEN
			Act_OpsRst;
		END_IF

	ELSIF eStatus <> Error THEN
		sStepTxt	:= 'Stop';
	ELSE
		sStepTxt	:= 'Error';
	END_IF

	//Reset
	IF EDGENEG(p_bRun) OR EDGEPOS(eStatus = Error) THEN
		Act_OpsInitial;
		Act_OpsRst;
	END_IF

	//Reset Error
	IF (eStatus = Error) AND bRstErr THEN
		eStatus		:= Idle;
		udiStatus	:= 0;
	END_IF

	//Always Run & Update
	IF p_bBufferMagPresent1 = FALSE
		OR (EDGENEG(p_bMcParamMagAWDis) AND p_tyBufferStat1.bBffrMty)
		THEN
		bMagAWDone	:= FALSE;

	END_IF

	IF (EDGENEG(p_bMcParamMagAWDis) AND p_tyBufferStat1.bBffrMty = FALSE)
		THEN
			bMagExitedWait:= TRUE;
			bNewMagVerified := FALSE;
	END_IF

//	IF (EDGENEG(p_bMcParamAutoRcpDis) OR EDGEPOS(p_bMcParamAutoRcpDis))AND p_tyBufferStat3.bBffrMty = FALSE THEN
//		bMagExitedWait:= TRUE;
//		ePrevExitStep := MagConvULStepMagExitMnl;
//	END_IF
	//
	IF p_usiUIHcomModchanged <> usiPrevHcomModchanged THEN //Flush out Magazine
		ePrevExitStep := MagConvULStepMagExitMnl;
		usiPrevHcomModchanged := p_usiUIHcomModchanged;
	END_IF

	fbMagRemovedTm(IN:= p_bMagPresentSen = FALSE AND p_bMagEntrySen = FALSE AND p_bDIMagFixedClampSen = FALSE AND p_bBufferMagRemoved);
	IF fbMagRemovedTm.Q  THEN
		iMagMESAcptCond 	:= 0;
		bMagExitedWait := FALSE;
		ePrevExitStep := MagConvULStepNA;
	END_IF

END_ACTION
```

#### Act_InitGlobal.st
```iecst
(** 2019-04-16 **)
ACTION Act_InitGlobal:

	(* Always Change If Project Change *)

	//Pass Data To Link
	p_bLinkDIMagPresentSen1 ACCESS p_DIMagPresentSen1;
	p_bLinkMagConv2Clp1MtrIn ACCESS p_MagConv2Clp1MtrSigOnOrLToR;
	p_bLinkMagConv2Clp1MtrOut ACCESS p_MagConv2Clp1MtrDirOrRToL;
	p_bLinkDIMagPresentSen2 ACCESS p_DIMagPresentSen2;
	p_bLinkMagConv2Clp2MtrIn ACCESS p_MagConv2Clp2MtrSigOnOrLToR;
	p_bLinkMagConv2Clp2MtrOut ACCESS p_MagConv2Clp2MtrDirOrRToL;
	p_bLinkDIMagPresentSen3 ACCESS p_DIMagPresentSen3;
	p_bLinkMagConv2Clp3MtrIn ACCESS p_MagConv2Clp3MtrSigOnOrLToR;
	p_bLinkMagConv2Clp3MtrOut ACCESS p_MagConv2Clp3MtrDirOrRToL;

	p_bLinkFixedMagClampRS1 ACCESS p_DIMag1FixedClampRS;
	p_bLinkRmtMagClampRS1 ACCESS p_DIMag1RemoteClampRS;

	p_bLinkFixedMagClampRS2 ACCESS p_DIMag2FixedClampRS;
	p_bLinkRmtMagClampRS2 ACCESS p_DIMag2RemoteClampRS;

	p_bLinkFixedMagClampRS3 ACCESS p_DIMag3FixedClampRS;
	p_bLinkRmtMagClampRS3 ACCESS p_DIMag3RemoteClampRS;

	p_bLinkDIMagEntrySen ACCESS p_DIMagConvEntSen1;
	p_bLinkMcParamMagAutoDetTm ACCESS p_McParamMagAutoDetTm;
	p_bLinkNtParamMagModelAutoVerify ACCESS p_NtParamProjMagAutoVerifyPrep;
	p_bLinkMagRcpCurrRcpMagModel ACCESS p_MagRcpCurrRcpMagModel;

	p_bLinkNewMagVerified2 ACCESS p_OpsMagConvUL2NewMagVerified;
	p_bLinkNewMagVerified3 ACCESS p_OpsMagConvUL3NewMagVerified;

	p_eLinkMcParamMagExMode ACCESS p_McParamMagExMode;

	p_bMag1OrientationChkSen1	ACCESS p_DIMag1OrientChkSen1;

	//Magazine Height Detection
	p_bMagHeightDetSen1			ACCESS p_DIHighMagDetSen1;
	p_bMagHeightDetEn 			ACCESS p_MagRcpCurrRcpMagHeightChkEn;
	p_bMagHeightDetPrep			ACCESS p_NtParamProjMagHeightChkPrep;

	p_bProjLifTravMnlLoad ACCESS p_NtParamProjLifTravMnlLoad;

	//Pass Data To Internal Use
	p_udiRstErr ACCESS p_RstErrReset;
	p_bEn ACCESS p_NtParamProjMag1ConvPrep;
	p_bRun ACCESS p_OpsRun;
	p_bStop ACCESS p_OpsStop;
	p_bStep ACCESS p_OpsStep;

	p_sProgNm ACCESS p_NtParamOpsMagConvUL1ProgNm;
	p_bNtSettingsLoadDone ACCESS p_StartupNtSettingsLoadDone;

	pa_bMagDis ACCESS p_OpsTravLifULMagDis;
	pa_bMagRej ACCESS p_OpsTravLifULMagRej;
//	p_bUSAllow ACCESS p_Follower2USAllow;

	p_bNewMag ACCESS p_UINewMag1;
	p_bRlsMag ACCESS p_UIRlsMag1;

	p_bConvInitDone ACCESS p_OpsTravLifULInitDone;
	p_bConvHvBrd ACCESS p_PshrConvHvBrd;
	p_bConvGdBrd ACCESS p_PshrConvGdBrd;

	p_tyBufferStat1 ACCESS p_Buffer1BffrStat;
	p_tyBufferStat2 ACCESS p_Buffer2BffrStat;
	p_tyBufferStat3 ACCESS p_Buffer3BffrStat;

	p_bMagEntrySen ACCESS p_DIMagConvEntSen1;
	p_bMagEntrySen1 ACCESS p_DIMagConvEntSen1;
	p_bMagEntrySen2 ACCESS p_DIMagConvEntSen2;
	p_bMagEntrySen3 ACCESS p_DIMagConvEntSen3;

	p_bMagPresentSen ACCESS p_DIMagPresentSen1;
	p_bMagPresentSen1 ACCESS p_DIMagPresentSen1;
	p_bMagPresentSen2 ACCESS p_DIMagPresentSen2;
	p_bMagPresentSen3 ACCESS p_DIMagPresentSen3;

	p_bBufferMagPresent1 ACCESS p_Buffer1MagPresent;
	p_bBufferMagPresent2 ACCESS p_Buffer2MagPresent;
	p_bBufferMagPresent3 ACCESS p_Buffer3MagPresent;

	p_dtBufferMagPresentTm1 ACCESS p_Buffer1MagPresentTm;
	p_dtBufferMagPresentTm2 ACCESS p_Buffer2MagPresentTm;
	p_dtBufferMagPresentTm3 ACCESS p_Buffer3MagPresentTm;

	p_eBufferStat ACCESS p_Buffer1Stat;
	p_eBufferStatus ACCESS p_Buffer1Status;

	p_bBufferMagRemoved ACCESS p_Buffer1MagRemoved;
	p_bBufferMagRemoved1 ACCESS p_Buffer1MagRemoved;
	p_bBufferMagRemoved2 ACCESS p_Buffer2MagRemoved;
	p_bBufferMagRemoved3 ACCESS p_Buffer3MagRemoved;

	p_eMagConv2ClpStat ACCESS p_MagConv2Clp1Stat;
	p_eMagConv2ClpStatus ACCESS p_MagConv2Clp1Status;
	p_bMagConv2ClpHvMag ACCESS p_MagConv2Clp1HvMag;

	p_eUSSMEMAStat ACCESS p_USSMEMA1Stat;
	p_eUSSMEMAStatus ACCESS p_USSMEMA1Status;
	p_bUSSMEMATransporting ACCESS p_USSMEMA1Transporting;
	p_bUSSMEMAConvStart ACCESS p_USSMEMA1ConvStart;
	p_bUSSMEMAConvStop ACCESS p_USSMEMA1ConvStop;

	p_eAGVMagStat ACCESS p_AGVMag1Stat;
	p_eAGVMagStatus ACCESS p_AGVMag1Status;
	p_bAGVMagMcRunRdy ACCESS p_AGVMag1McRunRdy;
	p_tyAGVToDTMag ACCESS p_AGVTagAGVToDTMag;

	p_eSelClampCtrlStat ACCESS p_PneuNoSenSelClamp1Stat;
	p_eSelClampCtrlStatus ACCESS p_PneuNoSenSelClamp1Status;

	p_bOutShutterExtended ACCESS p_Pneu2SenOutShutterExtended;

	p_bDIMagConvHeightSen ACCESS p_DIMagConvHeightSen1;
	p_bDIMagConvSelUnclampRS ACCESS p_DIMag1SelUnclampRS;
	p_bDIMagConvCAB717Sen ACCESS p_DIMagConvCAB717MagSen1;
	p_bDIMagConvSmallSen ACCESS p_DIMagConvSmallMagSen1;
	p_bDIMagConvLargeSen ACCESS p_DIMagConvLargeMagSen1;
	p_bDIOutShutterClosedRS ACCESS p_DIOutShutterCloseRS;

	p_eNtParamProjMagBuffferActLoad	ACCESS p_NtParamProjMagBuffferActLoad;

	p_eSafetyBarStat ACCESS p_Pneu2SMag1SafetyBarStat;
	p_eSafetyBarStatus ACCESS p_Pneu2SMag1SafetyBarStatus;
	p_bSafetyBarExtended ACCESS p_Pneu2SMag1SafetyBarExtended;
	p_bSafetyBarRetracted ACCESS p_Pneu2SMag1SafetyBarRetracted;

	p_eMagAWEngageStat ACCESS p_Pneu2SMag1AWEngageStat;
	p_eMagAWEngageStatus ACCESS p_Pneu2SMag1AWEngageStatus;

	p_eMagAWStat ACCESS p_MagAWOpen1Stat;
	p_eMagAWStatus ACCESS p_MagAWOpen1Status;
	p_bMagAWEngaging ACCESS p_MagAWOpen1Engaging;
	p_bMagAWErr ACCESS p_MagAWOpen1AxisErr;
	p_bMagAWOpenLimit ACCESS p_MagAWOpen1OpenSen;
	p_bMagAWCloseLimit ACCESS p_MagAWOpen1CloseSen;

	//USSOT
	p_eUSSOTStat ACCESS p_USSOT1Stat;
	p_eUSSOTStatus ACCESS p_USSOT1Status;
	p_bUSSOTTransporting ACCESS p_USSOT1Transporting;
	p_bUSSOTConvStart ACCESS p_USSOT1ConvStart;
	p_bUSSOTConvStop ACCESS p_USSOT1ConvStop;
	p_bUSSOTUSRdy ACCESS p_USSOT1USRdy;
	p_bUSSOTUSLargeMagRdy ACCESS p_USSOT1USLargeMagRdy;

	//DSSOT
	p_eDSSOTStat ACCESS p_DSSOT1Stat;
	p_eDSSOTStatus ACCESS p_DSSOT1Status;
	p_bDSSOTConvStart ACCESS p_DSSOT1ConvStart;
	p_bDSSOTConvStop ACCESS p_DSSOT1ConvStop;

	p_bOpsTravLifExitBrd ACCESS p_OpsTravLifULExitBrd;
	p_bOpsTravLifMov ACCESS p_OpsTravLifULTravLifMov;

	p_bSelfTest ACCESS p_OpsTravLifULSelfTest;

	p_bMcParamMagAWDis ACCESS p_McParamMagAWDis;

	p_bDISOTRcv ACCESS p_DISOT1Receive;
	p_bDISOTAGVReady ACCESS p_DISOT1Ready;

	p_eConvStat ACCESS p_PshrConvStat;
	p_eConvStatus ACCESS p_PshrConvStatus;

	p_eSafetyBarStat ACCESS p_Pneu2SMag1SafetyBarStat;
	p_eSafetyBarStatus ACCESS p_Pneu2SMag1SafetyBarStatus;
	p_bSafetyBarExtended ACCESS p_Pneu2SMag1SafetyBarExtended;
	p_bSafetyBarRetracted ACCESS p_Pneu2SMag1SafetyBarRetracted;

	p_sProdRcpCurrRcp1Name ACCESS p_ProdRcpCurrRcp1Nm;
	p_sProdRcpCurrRcp2Name ACCESS p_ProdRcpCurrRcp2Nm;

	p_bOpsTravLifErrCmdUnclmp ACCESS p_OpsTravLifWChkErrCmdUnclmp1;

	p_bNtParamAutoRcpPrep ACCESS p_NtParamAutoRcpPrep ;
	p_bMcParamAutoRcpDis  ACCESS p_McParamAutoRcpDisable;

	pa_bMagChangeOverBlk ACCESS p_AutoRcpbMagChangeOverBlk;
	p_bMagPropDiffBlk ACCESS p_AutoRcpbMag1PropDiffBlk;
	p_bChgMagWidth ACCESS p_AutoRcpbMag1WidthChg;
	p_bChgMagSlot ACCESS p_AutoRcpbMag1SlotChg;

	p_bMagOrientChkSenPrep ACCESS p_NtParamProjMagOrientChkSenPrep;
	p_bDIMagFixedClampSen ACCESS p_DIMag1FixedClampSen;

	p_eCustomerReq ACCESS p_NtParamCustomerReq;
	//For Siemen
	p_tyResponseFromMES ACCESS p_TagFromMesMagConv1;
	p_bOpsTravLifAllwExitMag ACCESS p_OpsTravLifAllwExitMag1;
	p_diMcParamMESResponseTO ACCESS p_McParamMESResponseTO;
	p_bMcParamMESEn ACCESS p_McParamMESEn;
	p_bAutoRcpForceExitMag ACCESS p_AutoRcpForceExitMag; //for switching Product
	p_dtCurrDT ACCESS p_TimeCurrDT;
	p_dtOpsMagConvUL2AcptTm ACCESS p_OpsMagConvUL2AcptTm;
	p_dtOpsMagConvUL3AcptTm ACCESS p_OpsMagConvUL3AcptTm;
	p_iOpsMagConvUL2MESAcptCond ACCESS p_OpsMagConvUL2MESAcptCond;
	p_iOpsMagConvUL3MESAcptCond ACCESS p_OpsMagConvUL3MESAcptCond;
	p_bOpsMagConvUL2MagExitedWait ACCESS p_OpsMagConvUL2MagExitedWait;
	p_bOpsMagConvUL3MagExitedWait ACCESS p_OpsMagConvUL3MagExitedWait;

	//Manual Flush when different Horizontal Com Mod
	p_usiUIHcomModchanged ACCESS p_UIHcomModchanged;
	(* Always Change If Project Change *)
	p_bNtParamAutoRcpF1ArbitraryType ACCESS p_NtParamAutoRcpF1ArbitraryType;
END_ACTION
```

#### Act_Initial.st
```iecst
(** 2019-01-20 **)
ACTION Act_Initial:

END_ACTION
```

#### Act_InitLocal.st
```iecst
(** 2019-04-16 **)
ACTION Act_InitLocal:

	//Input Reference Link To Local Variable
	p_udiRstErr ACCESS ADR(udiRstErr);
	p_bEn ACCESS ADR(bEn);
	p_bDis ACCESS ADR(bDis);
	p_bRun ACCESS ADR(bRun);
	p_bStop ACCESS ADR(bStop);
	p_bStep ACCESS ADR(bStep);

	p_sProgNm ACCESS ADR(sProgNm);
	p_bNtSettingsLoadDone ACCESS ADR(bNtSettingsLoadDone);

	p_usiMagConv ACCESS ADR(usiMagConv);
	p_bInfoEn ACCESS ADR(bInfoEn);

	pa_bMagDis ACCESS ADR(a_bMagDis);
	pa_bMagRej ACCESS ADR(a_bMagRej);
	p_bUSAllow ACCESS ADR(bUSAllow);

	p_bAllwChgWidth  ACCESS ADR(bAllwChgWidth);
	p_bAllwChgSlot ACCESS ADR(bAllwChgSlot);

	p_bNewMag ACCESS ADR(bNewMag);
	p_bRlsMag ACCESS ADR(bRlsMag);

	p_bConvInitDone ACCESS ADR(bConvInitDone);
	p_bConvHvBrd ACCESS ADR(bConvHvBrd);
	p_bConvGdBrd ACCESS ADR(bConvGdBrd);

	p_tyBufferStat1 ACCESS ADR(tyBufferStat1);
	p_tyBufferStat2 ACCESS ADR(tyBufferStat2);
	p_tyBufferStat3 ACCESS ADR(tyBufferStat3);

	p_bMagClampRS1 ACCESS ADR(bMagClampRS1);
	p_bMagClampRS2 ACCESS ADR(bMagClampRS2);
	p_bMagClampRS3 ACCESS ADR(bMagClampRS3);

	p_bMagEntrySen1 ACCESS ADR(bMagEntrySen1);
	p_bMagEntrySen2 ACCESS ADR(bMagEntrySen2);
	p_bMagEntrySen3 ACCESS ADR(bMagEntrySen3);

	p_bMagPresentSen1 ACCESS ADR(bMagPresentSen1);
	p_bMagPresentSen2 ACCESS ADR(bMagPresentSen2);
	p_bMagPresentSen3 ACCESS ADR(bMagPresentSen3);

	p_bBufferMagPresent1 ACCESS ADR(bBufferMagPresent1);
	p_bBufferMagPresent2 ACCESS ADR(bBufferMagPresent2);
	p_bBufferMagPresent3 ACCESS ADR(bBufferMagPresent3);

	p_dtBufferMagPresentTm1 ACCESS ADR(dtBufferMagPresentTm1);
	p_dtBufferMagPresentTm2 ACCESS ADR(dtBufferMagPresentTm2);
	p_dtBufferMagPresentTm3 ACCESS ADR(dtBufferMagPresentTm3);

	p_eBufferStat ACCESS ADR(eBufferStat);
	p_eBufferStatus ACCESS ADR(eBufferStatus);

	p_eMagConv2ClpStat ACCESS ADR(eMagConv2ClpStat);
	p_eMagConv2ClpStatus ACCESS ADR(eMagConv2ClpStatus);
	p_bMagConv2ClpHvMag ACCESS ADR(bMagConv2ClpHvMag);

	p_eUSSMEMAStat ACCESS ADR(eUSSMEMAStat);
	p_eUSSMEMAStatus ACCESS ADR(eUSSMEMAStatus);
	p_bUSSMEMATransporting ACCESS ADR(bUSSMEMATransporting);
	p_bUSSMEMAConvStart ACCESS ADR(bUSSMEMAConvStart);
	p_bUSSMEMAConvStop ACCESS ADR(bUSSMEMAConvStop);

	p_eAGVMagStat ACCESS ADR(eAGVMagStat);
	p_eAGVMagStatus ACCESS ADR(eAGVMagStatus);
	p_bAGVMagMcRunRdy ACCESS ADR(bAGVMagMcRunRdy);
	p_tyAGVToDTMag ACCESS ADR(tyAGVToDualMag);

	p_dtOpsMagConvUL1AcptTm ACCESS ADR(dtMagConvAcptTm);
	p_iOpsMagConvUL1MESAcptCond ACCESS ADR(iMagMESAcptCond);
END_ACTION
```

#### Act_Link.st
```iecst
(** 2018-12-11 **)
ACTION Act_Link:

	//Clamp RS
	p_bMagClampRS1 		:= (p_bLinkFixedMagClampRS1 AND p_bLinkRmtMagClampRS1) OR bNewMagVerified;
	p_bMagClampRS2		:= (p_bLinkFixedMagClampRS2 AND p_bLinkRmtMagClampRS2) OR p_bLinkNewMagVerified2;
	p_bMagClampRS3		:= (p_bLinkFixedMagClampRS3 AND p_bLinkRmtMagClampRS3) OR p_bLinkNewMagVerified3;

	//Mag Exchange Mode
	CASE p_eLinkMcParamMagExMode OF
		McSetMagXcAutoManMode:
			bMagManEx := TRUE;
			bMagAutoEx := TRUE;

		McSetMagXcAutoMode:
			bMagManEx := FALSE;
			bMagAutoEx := TRUE;

		McSetMagXcManMode:
			bMagManEx := TRUE;
			bMagAutoEx := FALSE;

	END_CASE

	//New magazine auto detection at inlet sensor
	fbMagAutoDetTm(IN := p_bLinkDIMagEntrySen OR p_bLinkDIMagPresentSen1, PT := DINT_TO_TIME(p_bLinkMcParamMagAutoDetTm));
	IF fbMagAutoDetTm.Q AND bMagManEx THEN
		bNewMagAutoDetected := TRUE;
	ELSE
		bNewMagAutoDetected := FALSE;
	END_IF

	IF p_bLinkNtParamMagModelAutoVerify THEN
		IF p_bLinkMagRcpCurrRcpMagModel = 0  //CAB706.2
			AND p_bDIMagConvHeightSen = TRUE
			AND p_bDIMagConvSelUnclampRS = FALSE
			AND p_bDIMagConvCAB717Sen = FALSE
			AND p_bDIMagConvSmallSen
			AND ((NOT p_bMagAWCloseLimit AND NOT  p_bMagAWOpenLimit) OR p_tyBufferStat1.bBffrMty = FALSE)
			THEN
			bNewMagVerified:= TRUE;

		ELSIF  p_bLinkMagRcpCurrRcpMagModel = 1 //CAB716.2
			AND p_bDIMagConvHeightSen = FALSE
			AND p_bDIMagConvSelUnclampRS = FALSE
			AND p_bDIMagConvCAB717Sen = FALSE
			AND p_bDIMagConvSmallSen
			AND ((NOT p_bMagAWCloseLimit AND NOT  p_bMagAWOpenLimit) OR p_tyBufferStat1.bBffrMty = FALSE)
			THEN
			bNewMagVerified:= TRUE;

		ELSIF  p_bLinkMagRcpCurrRcpMagModel = 2 //CAB717.2
			AND p_bDIMagConvHeightSen = FALSE
			AND p_bDIMagConvSelUnclampRS
			AND p_bDIMagConvCAB717Sen
			AND p_bDIMagConvLargeSen
			AND ((NOT p_bMagAWCloseLimit AND NOT  p_bMagAWOpenLimit) OR p_tyBufferStat1.bBffrMty = FALSE)
			THEN
			bNewMagVerified:= TRUE;
		ELSE
			bNewMagVerified:= FALSE;
		END_IF
	ELSE
		bNewMagVerified:= TRUE;
	END_IF

	IF p_bLinkMagRcpCurrRcpMagModel = 3 THEN
		bCAB703		:= TRUE;
		bFIXMag		:= FALSE;
	ELSIF p_bLinkMagRcpCurrRcpMagModel = 4 THEN
		bCAB703		:= FALSE;
		bFIXMag		:= TRUE;
	END_IF

	bAIVInPos := p_tyAGVToDTMag.bVEHInPos1 OR p_bDISOTRcv;

	IF p_bBufferMagRemoved THEN
		bManualUnloadMag := FALSE;
	END_IF

	IF bAutoRcpEn THEN
		//p_bNtParamAutoRcpF1ArbitraryType disable the use of AutoRcp MagSlot & Width Change Function
		p_bUSAllow :=  ( NOT(p_bNtParamAutoRcpF1ArbitraryType) AND NOT(p_bMagPropDiffBlk) ) AND
		(p_bNtParamAutoRcpF1ArbitraryType AND p_sProdRcpCurrRcp1Name = p_sProdRcpCurrRcp2Name)	;
		p_bAllwChgWidth := p_bChgMagWidth AND NOT(p_bNtParamAutoRcpF1ArbitraryType);
		p_bAllwChgSlot	:= p_bChgMagSlot AND NOT(p_bNtParamAutoRcpF1ArbitraryType);
	ELSE
		p_bUSAllow := p_sProdRcpCurrRcp1Name = p_sProdRcpCurrRcp2Name;
	END_IF

END_ACTION
```

#### Init.st
```iecst
(** 2019-03-25 **)
PROGRAM _INIT

	(* Always Change If Project Change *)

	//Physical Configuration
	usiMagConv	:= 1;
	bInfoEn		:= TRUE;

	//Pass Address To Global Address For External Use
	//Action, State & Status

	//Alarm
	p_OpsMagConvUL1AlmData	:= ADR(tyAlmData);
	p_OpsMagConvUL1AlmData1	:= ADR(tyAlmData1);

	//Output
	p_OpsMagConvUL1StepTxt	:= ADR(sStepTxt);
	p_OpsMagConvUL1Paused	:= ADR(bPaused);

	p_OpsMagConvUL1BufferAct		:= ADR(eBufferAct);
	p_OpsMagConvUL1MagConv2ClpAct	:= ADR(eMagConv2ClpAct);
	p_OpsMagConvUL1USSMEMAAct		:= ADR(eUSSMEMAAct);
	p_OpsMagConvUL1AGVMagAct		:= ADR(eAGVMagAct);

	p_OpsMagConvUL1InitDone				:= ADR(bOpsInitDone);
	p_OpsMagConvUL1MagBffrAvl			:= ADR(bMagBffrAvl);
	p_OpsMagConvUL1NewMagAllw			:= ADR(bNewMagAllw);
	p_OpsMagConvUL1RlsMagAllw			:= ADR(bRlsMagAllw);
	p_OpsMagConvUL1EjectMESStep			:= ADR(bEjectMESStep); //MES
	p_OpsMagConvUL1EjectMagNotAllw		:= ADR(bEjectMagNotAllw); //MES
	p_OpsMagConvUL1StepMagExitedWait	:= ADR(bStepMagExitedWait);
	p_OpsMagConvUL1StepUSCom			:= ADR(bStepMagUSCom);
	p_OpsMagConvUL1StepBffrLoad			:= ADR(bStepMagBffrLoad);
	p_OpsMagConvUL1StepPLCGrab			:= ADR(bStepPLCGrab);

	p_OpsMagConvUL1StepSelClampCtrl		:= ADR(eSelClampCtrl);
	p_OpsMagConvUL1NewMagVerified		:= ADR(bNewMagVerified);
	p_OpsMagConvUL1MagFullExit			:= ADR(bStepMagFullExit);
	p_OpsMagConvUL1IncorrectMagModel    := ADR(bIncorrectMagazineModel);
	p_OpsMagConvUL1MagSizeL    			:= ADR(bMagSizeLarge);

	p_OpsMagConvUL1SafetyBarAct			:= ADR(eSafetyBarAct);
	p_OpsMagConvUL1MagAWEngageAct		:= ADR(eMagAWEngageAct);
	p_OpsMagConvUL1MagAWAct				:= ADR(eMagAWAct);

	p_OpsMagConvUL1USSOTAct				:= ADR(eUSSOTAct);
	p_OpsMagConvUL1DSSOTAct				:= ADR(eDSSOTAct);

	p_OpsAGVCommRdy1					:= ADR(bAGVComm1Rdy);

	p_OpsMagConvUL1MsgReq				:= ADR(tyOpConMsgReq);

	p_OpsMagConvUL1UnclmpDone			:= ADR(bPneuUnclmpDone);
	p_OpsMagConvUL1MagAllwGo			:= ADR(udiMagAllwGo);

	p_OpsMagConvUL1ReadRFID				:= ADR(bReadRFID);
	p_OpsMagConvUL1WriteRFID			:= ADR(bWriteRFID);
	p_OpsMagConvUL1AWDone			 	:= ADR(bStepOpsMagAWDone);
	p_OpsMagConvUL1SlotUpdtDone			:= ADR(bStepOpsPitchUpdated);
	(* Always Change If Project Change *)

	p_OpsMagConvUL1AcptTm				:= ADR(dtMagConvAcptTm);
	p_OpsMagConvUL1MESAcptCond 			:= ADR(iMagMESAcptCond);
	p_OpsMagConvUL1MagExitedWait 		:= ADR(bMagExitedWait);

	//Mute Buzzer for Bosch China
	p_OpsMagConvUL1TLMuteBuzz			:= ADR(bTLMuteBuzzer);
	p_OpsMagConvUL1MagFullInfo			:=ADR(bMagFullInfo);

END_PROGRAM
```

#### Program Logical/Operations/MagConv_StationaryPlat/OpsMagConvUL1/Sequence

##### Act_OpsInfo.st
```iecst
ACTION Act_OpsInfo:

	//Reset
	udiStatus1	:= 0;
//	udiStatus2	:= 0;
	IF p_bInfoEn = TRUE THEN

			//Magazine Not Present
			a_bMagAllwMagPresent[1]	:= p_bBufferMagRemoved1 = FALSE;
			a_bMagAllwMagPresent[2]	:= p_bBufferMagRemoved2 = FALSE;
			a_bMagAllwMagPresent[3]	:= p_bBufferMagRemoved3 = FALSE;

			FOR udi := 1 TO 3 DO
				IF pa_bMagDis[udi] = FALSE AND a_bMagAllwMagPresent[udi] = TRUE THEN
					EXIT;
				END_IF
			END_FOR

			IF udi = 4 THEN
				IF eOpsStep > MagConvULStepInitMagConv OR eOpsStep = MagConvULStepMagUSComm THEN
					udiStatus1	:= 10000;
				END_IF
			END_IF

			//Magazine Is Full
			a_tyMagAllwBffrStat[1]	:= p_tyBufferStat1;
			a_tyMagAllwBffrStat[2]	:= p_tyBufferStat2;
			a_tyMagAllwBffrStat[3]	:= p_tyBufferStat3;

			FOR udi := 1 TO 3 DO
				IF pa_bMagDis[udi] = FALSE AND pa_bMagRej[udi] = TRUE THEN
					EXIT;
				END_IF
			END_FOR
			FOR udi1 := 1 TO 3 DO
				IF pa_bMagDis[udi1] = FALSE AND a_bMagAllwMagPresent[udi1] = TRUE AND a_tyMagAllwBffrStat[udi1].bBffrFull = TRUE THEN
					IF p_eCustomerReq = NA  OR (udi < 4 AND p_eCustomerReq = Bosch_China) THEN //Reject Mode Still
						udiStatus1	:= 10001 + (udi1 - 1);
						bTLMuteBuzzer := FALSE;
						EXIT;
					ELSIF (p_eCustomerReq = Bosch_China )  THEN
						bTLMuteBuzzer := TRUE;
						udiStatus1	:= 10001 + (udi1 - 1);
						FOR udi2 := 1 TO 3 DO
							IF udi2 <> udi1 THEN
								 IF pa_bMagDis[udi2] = FALSE AND a_bMagAllwMagPresent[udi2] = TRUE AND a_tyMagAllwBffrStat[udi2].bBffrFull = TRUE  THEN
									udiStatus1	:= 10001 + (udi2 - 1);
									EXIT;
								END_IF
							END_IF
						END_FOR
					END_IF
				END_IF
			END_FOR
			//when Magazine require to check this condition
			IF udiStatus1 <= 10004 AND udiStatus1<> 10000 THEN
				bMagFullInfo := TRUE;
			ELSE
				bMagFullInfo := FALSE;
			END_IF
			//Insert Good / Bad Magazine
			IF p_bConvInitDone = TRUE AND p_bConvHvBrd = TRUE THEN

				FOR udi := 1 TO 3 DO
					IF pa_bMagDis[udi] = FALSE AND pa_bMagRej[udi] = TRUE THEN
						EXIT;
					END_IF
				END_FOR

				IF udi < 4 THEN
					//Reject Mode
					IF p_bConvGdBrd = TRUE THEN
						//Good Board Exist
						FOR udi1 := 1 TO 3 DO
							IF pa_bMagDis[udi1] = FALSE AND a_bMagAllwMagPresent[udi1] = TRUE AND pa_bMagRej[udi1] = FALSE THEN
								EXIT;
							END_IF
						END_FOR

						IF udi1 = 4 THEN
							udiStatus1	:= 10004;
						END_IF

					ELSE
						//Bad Board Exist
						FOR udi1 := 1 TO 3 DO
							IF pa_bMagDis[udi1] = FALSE AND a_bMagAllwMagPresent[udi1] = TRUE AND pa_bMagRej[udi1] = TRUE THEN
								EXIT;
							END_IF
						END_FOR

						IF udi1 = 4 THEN
							udiStatus1	:= 10005;
						END_IF

					END_IF

				ELSE
					//Non-Reject Mode
					FOR udi1 := 1 TO 3 DO
						IF pa_bMagDis[udi1] = FALSE AND a_bMagAllwMagPresent[udi1] = TRUE THEN
							EXIT;
						END_IF
					END_FOR

					IF udi1 = 4 THEN
						udiStatus1	:= 10004;
					END_IF

				END_IF

			END_IF
	END_IF

		//Magazine Verification Warning

	IF fbMagRemovedTm.Q OR bNewMagVerified THEN
		bNewMagVerifyStarted := FALSE;
	END_IF

	fbVerifyWarningDelay(IN:= bNewMagVerifyStarted AND bNewMagVerified = FALSE AND bStepMagVerification = FALSE);

	IF fbVerifyWarningDelay.Q AND p_tyBufferStat1.bBffrFull = FALSE THEN
		IF   (p_bMagAWCloseLimit OR  p_bMagAWOpenLimit) AND p_tyBufferStat1.bBffrMty THEN
			bLimitSenActivated := TRUE;
			udiStatus1	:= 10010;
		ELSIF bLimitSenActivated THEN
			udiStatus1	:= 10010;
		ELSIF bManualUnloadMag = FALSE THEN
			CASE p_bLinkMagRcpCurrRcpMagModel OF
			0: //CAB706.2
				IF bWrongHeight THEN
					udiStatus1	:= 10007;
				ELSIF p_bDIMagConvHeightSen = FALSE THEN
					bWrongHeight := TRUE;

				ELSIF bWrongWidth THEN
					udiStatus1	:= 10006;
				ELSIF p_bDIMagConvSelUnclampRS
					OR p_bDIMagConvCAB717Sen
					OR p_bDIMagConvSmallSen = FALSE
					THEN
					bWrongWidth := TRUE;

				END_IF

			1: //CAB716.2
				IF bWrongHeight THEN
					udiStatus1	:= 10007;
				ELSIF p_bDIMagConvHeightSen = TRUE THEN
					bWrongHeight := TRUE;

				ELSIF bWrongWidth THEN
					udiStatus1	:= 10006;
				ELSIF p_bDIMagConvSelUnclampRS
					OR p_bDIMagConvCAB717Sen
					OR p_bDIMagConvSmallSen = FALSE
					THEN
					bWrongWidth := TRUE;

				END_IF

			2: //CAB717.2
				IF bWrongHeight THEN
					udiStatus1	:= 10007;
				ELSIF p_bDIMagConvHeightSen THEN
					bWrongHeight := TRUE;

				ELSIF bWrongWidth THEN
					udiStatus1	:= 10006;
				ELSIF p_bDIMagConvSelUnclampRS = FALSE
					OR p_bDIMagConvCAB717Sen = FALSE
					OR p_bDIMagConvLargeSen
					THEN
					bWrongWidth := TRUE;

				END_IF

			END_CASE
		ELSIF bManualUnloadMag THEN
			udiStatus1	:= 10008;
		END_IF
	ELSIF udiStatus1 <> 10006
		AND udiStatus1 <> 10007
		AND p_tyBufferStat1.bBffrFull = FALSE
		AND bStepMagExitedWait
		AND p_bLocalMagEntrySen
		THEN
		udiStatus1	:= 10008;
		bManualUnloadMag := TRUE;

	ELSE
		bLimitSenActivated := FALSE;
		bWrongHeight := FALSE;
		bWrongWidth	:= FALSE;
	END_IF

	bIncorrectMagazineModel := udiStatus1 = 10006 OR udiStatus1 = 10007;

	//@@@@@@@@@@@@@@@@@@@@ opCon @@@@@@@@@@@@@@@@@@@@@@@@@@@@@@@@@@@@@@@@@@@@@@@@@@@@
	IF udiStatus1 = 10000 THEN
		fbIdleTm (IN:= TRUE);
		IF fbIdleTm.Q THEN
			fbIdleTm (IN:= FALSE);
			bPartMissingStarted := TRUE;
			tyOpConMsgReq := OpConMsgTypePartMissingStarted;
		END_IF
	ELSIF bPartMissingStarted AND (p_bMagPresentSen1 OR p_bMagPresentSen2 OR p_bMagPresentSen3) THEN
		bPartMissingStarted := FALSE;
		tyOpConMsgReq := OpConMsgTypePartMissing;
	ELSE
		fbIdleTm (IN:= FALSE);
	END_IF

	//----------------------------Siemens MES -------------------------------------//
	IF (udiStatus1 = 0 OR udiStatus1 = 10008) AND (p_eCustomerReq = Siemens OR p_eCustomerReq = We_Fabricate ) THEN
		IF eOpsStep = MagConvULStepMagEntMESStdByChk  THEN
			IF NOT(fbReadRFIDTO.Q) THEN //Reading RFID
				udiStatus1 := 10012;
			ELSE   //Reading RFID Time Out,Press Release Then Exit
				udiStatus1 := 10013;
			END_IF
		ELSIF eOpsStep = MagConvULStepMagExtMESStdByChk   THEN//
			IF NOT(fbWriteRFIDTO.Q) THEN
				udiStatus1 := 10014;
			ELSE
				udiStatus1 := 10015;
			END_IF

		ELSIF (eOpsStep = MagConvULStepMagFullDSComm OR eOpsStep = MagConvULStepMagExitMnl OR eOpsStep = MagConvULStepMagExitedWait) AND iMagMESAcptCond < 0  THEN
			udiStatus1 := 10016; //Wrong Magazine Position 1
		END_IF
	END_IF
END_ACTION
```

##### Act_OpsInitial.st
```iecst
(** 2019-01-16 **)
ACTION Act_OpsInitial:

	eOpsStep		:= MagConvULStepNA;
	eGotoOpsStep	:= MagConvULStepInitMag;

	bOpsInitDone		:= FALSE;
	bMagBffrAvl			:= FALSE;
	bNewMagAllw			:= FALSE;
	bRlsMagAllw			:= FALSE;
	bStepMagExitedWait	:= FALSE;
	bAGVComm1Rdy		:= FALSE;

END_ACTION
```

##### Act_OpsRst.st
```iecst
(** 2019-03-25 **)
ACTION Act_OpsRst:

	udiStatus1	:= 0;

	eBufferAct		:= BufferActIdle;
	eMagConv2ClpAct	:= MagConv2ClpActIdle;
	eUSSMEMAAct		:= SMEMAActIdle;
	eAGVMagAct		:= AGVMagActIdle;
	eSelClampCtrl	:= PneuActIdle;
	eSafetyBarAct	:= PneuActIdle;
	eMagAWEngageAct	:= PneuActIdle;
	eMagAWAct		:= MagAWActIdle;
	eDSSOTAct		:= SOTActIdle;
	eUSSOTAct		:= SOTActIdle;

	bNewMagVerified := FALSE;
	bNewMagVerifyStarted := FALSE;

	bPneuUnclmpDone		 := FALSE;
	bReadRFID := FALSE;
	bWriteRFID := FALSE;

//	fbWriteRFIDTO(IN:= FALSE);
END_ACTION
```

##### Act_OpsRun.st
```iecst
(** 2019-04-16 **)
ACTION Act_OpsRun:
	IF p_bOpsTravLifErrCmdUnclmp THEN //from travLif width chk error
		eMagConv2ClpAct :=	MagConv2ClpActStopClpr;

		IF (p_eMagConv2ClpStatus = Done AND p_eMagConv2ClpStat = MagConv2ClpActStopClpr) THEN

			eMagConv2ClpAct	:= MagConv2ClpActIdle;
			bPneuUnclmpDone := TRUE; //To TravLifUL
		END_IF
	END_IF

	Act_LogStep;

	IF eGotoOpsStep <> eOpsStep THEN

		fbWrongMagTm(IN:= FALSE);
		fbReadRFIDTO(IN:= FALSE);
		fbWriteRFIDTO(IN:= FALSE);
		CASE eGotoOpsStep OF
			MagConvULStepBffrStatChk:  //For Siemen, Enter Condition
				IF ((p_eCustomerReq = Siemens OR p_eCustomerReq = We_Fabricate)AND p_bMcParamMESEn) AND eOpsStep = MagConvULStepVerifyMag THEN
					IF ePrevStepBeforeMESStdBy = MagConvULStepMagExitMnl OR ePrevStepBeforeMESStdBy = MagConvULStepMagExitClampCtrl THEN
						eGotoOpsStep		:= MagConvULStepMagExtMESStdByChk;
						eOpsStep			:= MagConvULStepMagExtMESStdByChk;
					ELSIF  iMagMESAcptCond > 0 THEN
						eGotoOpsStep		:= MagConvULStepBffrStatChk;
						eOpsStep			:= MagConvULStepBffrStatChk;
					ELSIF iMagMESAcptCond < 0 THEN
						eGotoOpsStep		:= MagConvULStepMagExitClampCtrl;
						eOpsStep			:= MagConvULStepMagExitClampCtrl;
					ELSIF iMagMESAcptCond = 0 THEN
						eGotoOpsStep		:= MagConvULStepMagEntMESStdByChk;
						eOpsStep			:= MagConvULStepMagEntMESStdByChk;
					END_IF
				ELSE
					eOpsStep	:= eGotoOpsStep;
				END_IF
			MagConvULStepMagExitClampCtrl: //For Siemen, Bffr Full,Changover Mag, AGV Rdy,Reject Mag
				IF (p_eCustomerReq = Siemens AND p_bMcParamMESEn) AND (eOpsStep <> MagConvULStepMagExtMESStdByChk )
					AND (p_tyLocalBufferStat.bBffrFull OR pa_bMagChangeOverBlk[p_usiMagConv] = TRUE OR p_bDISOTAGVReady)
					AND NOT(iMagMESAcptCond < 0)THEN
					eOpsStep := MagConvULStepMagExtMESStdByChk;
					eGotoOpsStep := MagConvULStepMagExtMESStdByChk;
					ePrevStepBeforeMESStdBy := MagConvULStepMagExitClampCtrl;
				ELSE
					eOpsStep	:= eGotoOpsStep;
					ePrevStepBeforeMESStdBy	:= MagConvULStepNA;
				END_IF
			MagConvULStepMagExitMnl: //For Siemens, Manual Rls
				IF (p_eCustomerReq = Siemens AND p_bMcParamMESEn)
					AND (eOpsStep <> MagConvULStepMagExtMESStdByChk AND eOpsStep <> MagConvULStepMagFullDSComm
					AND eOpsStep <> MagConvULStepMagEntMESStdByChk AND eOpsStep <> MagConvULStepVerifyMag)
					 THEN
					eOpsStep := MagConvULStepMagExtMESStdByChk;
					eGotoOpsStep := MagConvULStepMagExtMESStdByChk;
					ePrevStepBeforeMESStdBy := MagConvULStepMagExitMnl;
				ELSE
//					sStepTxt	:= 'Waiting for Shutter Close';

//					IF p_bDIOutShutterClosedRS THEN
						eOpsStep	:= eGotoOpsStep;
						ePrevStepBeforeMESStdBy	:= MagConvULStepNA;
//					END_IF
				END_IF
			MagConvULStepSelClampCtrl:
				IF p_bMagOrientChkSenPrep THEN
					IF p_bMagHeightDetEn AND p_bMagHeightDetPrep THEN

						IF p_bMag1OrientationChkSen1 AND p_bMagHeightDetSen1 THEN // Magazine Type Check with height Detection Sensor
							eOpsStep := eGotoOpsStep;
						ELSE
							eMagConv2ClpAct :=	MagConv2ClpActStopClpr; //Unclamp First

							IF (p_eMagConv2ClpStatus = Done AND p_eMagConv2ClpStat = MagConv2ClpActStopClpr) THEN

								eMagConv2ClpAct	:= MagConv2ClpActIdle;

								eStatus		:= Error;
								udiStatus	:= 10011;	//Wrong Magazine Orientation Placed.
							END_IF
						END_IF

					ELSE

						IF p_bMag1OrientationChkSen1 AND NOT p_bMagHeightDetSen1 THEN //Without Check Height Detection Sensor
							eOpsStep := eGotoOpsStep;
						ELSE
							eMagConv2ClpAct :=	MagConv2ClpActStopClpr; //Unclamp First

							IF (p_eMagConv2ClpStatus = Done AND p_eMagConv2ClpStat = MagConv2ClpActStopClpr) THEN

								eMagConv2ClpAct	:= MagConv2ClpActIdle;

								eStatus		:= Error;
								udiStatus	:= 10011;	//Wrong Magazine Orientation Placed.
							END_IF
						END_IF

					END_IF
				ELSE
					eOpsStep	:= eGotoOpsStep;
				END_IF
			ELSE
				eOpsStep	:= eGotoOpsStep;

		END_CASE

	END_IF

	IF eOpsStep = eGotoOpsStep THEN

		IF bPaused = FALSE THEN

			CASE eOpsStep OF

				MagConvULStepInitMag:
					sStepTxt	:= 'Initializing Magazine';
					p_usiMagConv := 1;
					CASE p_usiMagConv OF
						1:
							p_tyLocalBufferStat ACCESS ADR(p_tyBufferStat1);
							p_bLocalMagEntrySen ACCESS ADR(p_bMagEntrySen1);
							p_bLocalBufferMagPresent ACCESS ADR(p_bBufferMagPresent1);
							p_dtLocalBufferMagPresentTm ACCESS ADR(p_dtBufferMagPresentTm1);
						2:
							p_tyLocalBufferStat ACCESS ADR(p_tyBufferStat2);
							p_bLocalMagEntrySen ACCESS ADR(p_bMagEntrySen2);
							p_bLocalBufferMagPresent ACCESS ADR(p_bBufferMagPresent2);
							p_dtLocalBufferMagPresentTm ACCESS ADR(p_dtBufferMagPresentTm2);
						3:
							p_tyLocalBufferStat ACCESS ADR(p_tyBufferStat3);
							p_bLocalMagEntrySen ACCESS ADR(p_bMagEntrySen3);
							p_bLocalBufferMagPresent ACCESS ADR(p_bBufferMagPresent3);
							p_dtLocalBufferMagPresentTm ACCESS ADR(p_dtBufferMagPresentTm3);
					END_CASE

//					IF bMagExitedWait THEN
//						eGotoOpsStep	:= MagConvULStepMagExitedWait;
//					ELSE
//						eGotoOpsStep	:= MagConvULStepInitMagConv;
//					END_IF
					IF p_bProjLifTravMnlLoad = FALSE THEN
						eGotoOpsStep	:= MagConvULStepInitAWPneu;
					ELSE
						eGotoOpsStep	:= MagConvULStepMagUSComm; //no roller
					END_IF

					bPaused	:= p_bStop OR p_bStep;

				MagConvULStepInitAWPneu:
					sStepTxt	:= 'Initializing Pneumatic';

					eSafetyBarAct	:= PneuActExt;
					eMagAWEngageAct	:= PneuActRet;

					IF (p_eSafetyBarStatus = Done AND p_eSafetyBarStat = PneuActExt) AND (p_eMagAWEngageStatus = Done AND p_eMagAWEngageStat = PneuActRet) THEN
						eSafetyBarAct	:= PneuActIdle;
						eMagAWEngageAct	:= PneuActIdle;
						IF bMagExitedWait AND  ePrevExitStep = MagConvULStepMagExitMnl THEN
							//	eDSSOTAct	:= SOTActRun;
							eGotoOpsStep		:= MagConvULStepMagExitedWait; //sucessful exited
						ELSIF ePrevExitStep = MagConvULStepMagExitMnl THEN
							eGotoOpsStep	:= MagConvULStepInitMagEnt; //halfway exiting, if magazine gone, init step
							//eGotoOpsStep	:= MagConvULStepMagExitMnl;
//						ELSIF ePrevExitStep = MagConvULStepMagExitClampCtrl THEN
//							eGotoOpsStep	:= MagConvULStepMagExitClampCtrl; //want to exit before clamping
						ELSE
							eGotoOpsStep	:= MagConvULStepInitMagConv;
						END_IF
					END_IF

				MagConvULStepInitMagEnt:
					sStepTxt	:= 'Initializing Magazine Conveyor';
					eMagConv2ClpAct	:= MagConv2ClpActInit;
					IF (p_eMagConv2ClpStatus = Done AND p_eMagConv2ClpStat = MagConv2ClpActInit) THEN
						eMagConv2ClpAct	:= MagConv2ClpActIdle;
						IF p_bMagConv2ClpHvMag = FALSE THEN
							eGotoOpsStep	:= MagConvULStepMagUSComm;
							ePrevExitStep 		:= MagConvULStepNA;
							iMagMESAcptCond 	:= 0;
						ELSE
							eGotoOpsStep	:= MagConvULStepInitMagFixClp;
						END_IF
					END_IF

				MagConvULStepInitMagFixClp:
					sStepTxt	:= 'Initializing Fixed Clamp';
					eMagConv2ClpAct	:= MagConv2ClpActFixClprClamp;
					IF (p_eMagConv2ClpStatus = Done AND p_eMagConv2ClpStat = MagConv2ClpActFixClprClamp) THEN
							eMagConv2ClpAct	:= MagConv2ClpActIdle;
							IF bMagAutoEx THEN
								eDSSOTAct	:= SOTActRun;
							ELSE
								eDSSOTAct	:= SOTActIdle;
							END_IF

							IF p_bDIMagConvCAB717Sen THEN
								bMagSizeLarge := TRUE;
							ELSE
								bMagSizeLarge := FALSE;
							END_IF
							eGotoOpsStep	:= MagConvULStepSelClampCtrl;
					END_IF

				MagConvULStepInitMagConv:
					sStepTxt	:= 'Initializing Magazine Conveyor';

					eMagConv2ClpAct	:= MagConv2ClpActInitStopClp;
					eSelClampCtrl := PneuActExt;

					IF (p_eMagConv2ClpStatus = Done AND p_eMagConv2ClpStat = MagConv2ClpActInitStopClp)
						AND (p_eSelClampCtrlStat = PneuActExt AND p_eSelClampCtrlStatus = Done)
						THEN
						eSelClampCtrl := PneuActIdle;
						eMagConv2ClpAct	:= MagConv2ClpActIdle;

						IF p_bMagConv2ClpHvMag = FALSE THEN
							eGotoOpsStep	:= MagConvULStepMagUSComm;
							ePrevExitStep 		:= MagConvULStepNA;
							iMagMESAcptCond 	:= 0;
						ELSE
							//	eGotoOpsStep	:= MagConvULStepBffrStatChk;
							eGotoOpsStep	:= MagConvULStepSelClampCtrl;
						END_IF

						bPaused	:= p_bStop OR p_bStep;
					END_IF

				MagConvULStepMagUSComm:
					sStepTxt	:= 'Communicating AIV And Ready For Transport In Magazine';

					eAGVMagAct	:= AGVMagActEnter;
					IF bMagAutoEx THEN
						eUSSOTAct	:= SOTActRun;
					ELSE
						eUSSOTAct	:= SOTActIdle;
					END_IF

					eDSSOTAct	:= SOTActIdle;
					bMagSizeLarge := FALSE;
					bMagExitedWait	:= FALSE;

					IF p_bSafetyBarExtended = FALSE THEN
						eGotoOpsStep	:= MagConvULStepSafetyBarExt;
					ELSIF p_bAGVMagMcRunRdy = TRUE OR p_bUSSOTTransporting= TRUE THEN
						eGotoOpsStep	:= MagConvULStepMagEnt;

					ELSIF p_bNewMag = TRUE OR bNewMagAutoDetected = TRUE THEN
						eAGVMagAct		:= AGVMagActIdle;
						eGotoOpsStep	:= MagConvULStepMagEntMnl;

					ELSE
						bPaused	:= p_bStop;

						IF bPaused = TRUE THEN
							eAGVMagAct	:= AGVMagActIdle;
							eUSSOTAct	:= SOTActIdle;
						END_IF

					END_IF

				MagConvULStepMagEnt:

					IF p_bUSSOTConvStart THEN
						sStepTxt	:= 'Conveyor Entering Magazine To End';
						eMagConv2ClpAct	:= MagConv2ClpActEntStopClp;

					ELSIF bNewMagAutoDetected = TRUE THEN
						eAGVMagAct			:= AGVMagActIdle;
						eGotoOpsStep		:= MagConvULStepMagEntMnl;

					ELSIF p_bUSSOTConvStop THEN
						sStepTxt	:= 'Conveyor Stopping';
						eMagConv2ClpAct	:= MagConv2ClpActStopClpr;
						IF (p_eMagConv2ClpStatus = Done AND p_eMagConv2ClpStat = MagConv2ClpActStopClpr) THEN
							eMagConv2ClpAct		:= MagConv2ClpActIdle;

						END_IF
					END_IF

					IF (p_eMagConv2ClpStatus = Done AND p_eMagConv2ClpStat = MagConv2ClpActEntStopClp) THEN
						eAGVMagAct			:= AGVMagActIdle;
						eMagConv2ClpAct		:= MagConv2ClpActIdle;
						eUSSOTAct			:= SOTActIdle;
						eGotoOpsStep		:= MagConvULStepSelClampCtrl;
						bPaused	:= p_bStop OR p_bStep;

					ELSE

					END_IF

				MagConvULStepMagEntMnl:
					sStepTxt	:= 'Magazine Conveyor Entering Magazine Manually';
					IF p_bProjLifTravMnlLoad = FALSE THEN
						eMagConv2ClpAct	:= MagConv2ClpActEntStopClp;
					ELSE
						eGotoOpsStep	:= MagConvULStepSelClampCtrl; //no roller
					END_IF

					IF p_eMagConv2ClpStatus = Done AND p_eMagConv2ClpStat = MagConv2ClpActEntStopClp THEN
						eMagConv2ClpAct	:= MagConv2ClpActIdle;
						//	eGotoOpsStep	:= MagConvULStepBffrStatChk;
							eGotoOpsStep	:= MagConvULStepSelClampCtrl;
						eUSSOTAct			:= SOTActIdle;
						eAGVMagAct			:= AGVMagActIdle;
						bPaused	:= p_bStop OR p_bStep;
					END_IF

				MagConvULStepSelClampCtrl:
					sStepTxt	:= 'Magazine Selection Control';
					bNewMagVerifyStarted := TRUE;

					CASE p_bLinkMagRcpCurrRcpMagModel OF
						0: //CAB706.2
							IF p_bDIMagConvCAB717Sen = FALSE THEN
								eSelClampCtrl := PneuActRet;
							END_IF

							eGotoOpsStep		:= MagConvULStepVerifyMag;

						1: //CAB716.2
							IF p_bDIMagConvCAB717Sen = FALSE THEN
								eSelClampCtrl := PneuActRet;
							END_IF

							eGotoOpsStep		:= MagConvULStepVerifyMag;

						2: //CAB717.2
							eSelClampCtrl := PneuActExt;

							eGotoOpsStep	:= MagConvULStepVerifyMag;

					END_CASE

					bPaused	:= p_bStop OR p_bStep;

				MagConvULStepVerifyMag: //Model Verificaiton
					sStepTxt	:= 'Magazine Model Verification';

					bNewMagVerifyStarted := TRUE;
					fbWrongMagTm(IN:= bNewMagVerified = FALSE);
					IF fbWrongMagTm.Q AND NOT bMagExitedWait THEN
						fbWrongMagTm(IN:= FALSE);
						eGotoOpsStep		:= MagConvULStepMagExitMnl;
					ELSIF ePrevExitStep = MagConvULStepMagExitMnl THEN
						eGotoOpsStep		:= MagConvULStepMagExitMnl;
					ELSIF ePrevExitStep = MagConvULStepMagExitClampCtrl THEN
						eGotoOpsStep		:= MagConvULStepMagExitClampCtrl;
					ELSIF bNewMagVerified  THEN
						eSelClampCtrl	:= PneuActIdle;

						eGotoOpsStep		:= MagConvULStepBffrStatChk; //to RFID scanning if applicable

					END_IF

					IF p_bDIMagConvCAB717Sen THEN
						bMagSizeLarge := TRUE;
					ELSE
						bMagSizeLarge := FALSE;
					END_IF

					IF p_bSelfTest THEN
						eGotoOpsStep	:= MagConvULStepMagCmp;
					END_IF

					bPaused	:= p_bStop OR p_bStep;
				MagConvULStepMagEntMESStdByChk:
					IF p_eCustomerReq = Siemens THEN
						sStepTxt	:= 'Read RFID Chk step';
					ELSE
						sStepTxt	:= 'Wait for MES feedback';
					END_IF
					bReadRFID := TRUE;
					fbReadRFIDTO(IN:= bReadRFID,PT := DINT_TO_TIME(p_diMcParamMESResponseTO));
					iMagMESAcptCond := (p_tyResponseFromMES.iAcceptCondition);
					IF p_tyResponseFromMES.iAcceptCondition > 0  THEN //Accept
						eGotoOpsStep := MagConvULStepBffrStatChk;
						dtMagConvAcptTm	:= p_dtCurrDT;
					ELSIF p_tyResponseFromMES.iAcceptCondition < 0  THEN//No Accept
						eGotoOpsStep	:= MagConvULStepMagExitClampCtrl;
					ELSIF fbReadRFIDTO.Q AND p_bRlsMag THEN
						sStepTxt	:= 'Wait for Read RFID';
						eGotoOpsStep := MagConvULStepMagExitMnl;
					END_IF
					IF eGotoOpsStep <> MagConvULStepMagEntMESStdByChk THEN
						bReadRFID := FALSE;
						fbReadRFIDTO(IN:= bReadRFID);
					END_IF
					bPaused	:= p_bStop OR p_bStep;
				MagConvULStepBffrStatChk:
					sStepTxt	:= 'Checking Buffer Status';

					IF p_eBufferStatus = Idle THEN

						IF p_tyLocalBufferStat.bBffrFull = TRUE
							//AND p_bOutShutterExtended
							THEN
							//	eGotoOpsStep	:= MagConvULStepMagFullDSComm;
							eGotoOpsStep	:= MagConvULStepMagExitClampCtrl;
						ELSE
		//	20210420		eGotoOpsStep	:= MagConvULStepMagCmp;
							eGotoOpsStep	:= MagConvULStepSafetyBarRet;
						END_IF

						bPaused	:= p_bStop OR p_bStep;

					END_IF

				MagConvULStepChkMag:

					sStepTxt	:= 'Checking Magazine Status';
//					IF p_bSafetyBarExtended = FALSE THEN
//							eGotoOpsStep	:= MagConvULStepSafetyBarExt;

//					ELSIF p_bMagPresentSen1 = TRUE THEN
					IF p_bMagPresentSen = TRUE THEN
						IF p_tyLocalBufferStat.bBffrMty = TRUE THEN
							//Buffer Empty
							IF  bAutoRcpEn THEN
								eGotoOpsStep	:= MagConvULStepMagCmp;
							ELSIF bMagAWDone = FALSE THEN
								eGotoOpsStep	:= MagConvULStepMagAWEngage;
//							ELSIF p_bSafetyBarRetracted = FALSE THEN
//								eGotoOpsStep	:= MagConvULStepSafetyBarRet;
							ELSE
								eGotoOpsStep	:= MagConvULStepMagCmp;
							END_IF

						ELSIF p_tyLocalBufferStat.bBffrFull = TRUE
						//	AND p_bOutShutterExtended
							THEN
							//Buffer Full

							IF p_bSafetyBarExtended = FALSE THEN
								eGotoOpsStep	:= MagConvULStepSafetyBarExt;
							ELSE
								eGotoOpsStep    := MagConvULStepMagExitClampCtrl;
							END_IF

						ELSE
							//Buffer Available
//							IF p_bSafetyBarRetracted = FALSE THEN
//								eGotoOpsStep	:= MagConvULStepSafetyBarRet;
//							ELSE
								eGotoOpsStep	:= MagConvULStepMagCmp;
//							END_IF

						END_IF

					ELSE

//						IF p_bSafetyBarExtended = FALSE THEN
//							eGotoOpsStep	:= MagConvULStepSafetyBarExt;
//						ELSE
							eGotoOpsStep	:= MagConvULStepMagUSComm;
//						END_IF

					END_IF

					bPaused	:= p_bStop OR p_bStep;

				MagConvULStepSafetyBarExt:
					sStepTxt	:= 'Extending Safety Bar';

					eSafetyBarAct	:= PneuActExt;

					IF p_eSafetyBarStatus = Done AND p_eSafetyBarStat = PneuActExt THEN
						eSafetyBarAct	:= PneuActIdle;
						eGotoOpsStep	:= MagConvULStepChkMag;

						bPaused	:= p_bStop OR p_bStep;
					END_IF

				MagConvULStepSafetyBarRet:
					sStepTxt	:= 'Retracting Safety Bar';

					eSafetyBarAct	:= PneuActRet;

					IF p_eSafetyBarStatus = Done AND p_eSafetyBarStat = PneuActRet THEN
						eSafetyBarAct	:= PneuActIdle;
					//	eGotoOpsStep	:= MagSetupULStepMagNBffrStatChk;
						eGotoOpsStep	:= MagConvULStepChkMag;

						bPaused	:= p_bStop OR p_bStep;
					END_IF

				MagConvULStepMagAWEngage:
					sStepTxt	:= 'Engaging Magazine Auto Width';

					eMagAWAct	:= MagAWActEngage;

					IF p_bMagAWEngaging = TRUE THEN
						eMagAWEngageAct	:= PneuActExt;
					END_IF

					IF (p_eMagAWStatus = Done AND p_eMagAWStat = MagAWActEngage) AND (p_eMagAWEngageStatus = Done AND p_eMagAWEngageStat = PneuActExt) THEN
						eMagAWAct		:= MagAWActIdle;
						eMagAWEngageAct	:= PneuActIdle;
						eGotoOpsStep	:= MagConvULStepMagAWHm;
						bPaused	:= p_bStop OR p_bStep;

					END_IF

				MagConvULStepMagAWHm:
					sStepTxt	:= 'Homing Magazine Auto Width';

					eMagAWAct	:= MagAWActHoming;

					IF p_eMagAWStatus = Done AND p_eMagAWStat = MagAWActHoming THEN
						eMagAWAct		:= MagAWActIdle;
						eGotoOpsStep	:= MagConvULStepMagAWMov;

					ELSIF p_bMagAWErr THEN

						eStatus			:= Error;
						udiStatus		:= 10009;
					END_IF

				MagConvULStepMagAWMov:
					sStepTxt	:= 'Moving Magazine Auto Width';

					eMagAWAct	:= MagAWActGoWidthOff;

					IF p_eMagAWStatus = Done AND p_eMagAWStat = MagAWActGoWidthOff THEN
						bMagAWDone		:= TRUE;
						eMagAWAct		:= MagAWActIdle;
						eGotoOpsStep	:= MagConvULStepMagAWDisengage;

						bPaused	:= p_bStop OR p_bStep;

					ELSIF p_bMagAWErr THEN

						eStatus			:= Error;
						udiStatus		:= 10009;
					END_IF

				MagConvULStepMagAWDisengage:
					sStepTxt	:= 'Disengaging Magazine Auto Width';

					eMagAWEngageAct	:= PneuActRet;

					IF p_eMagAWEngageStatus = Done AND p_eMagAWEngageStat = PneuActRet THEN
						eMagAWEngageAct	:= PneuActIdle;

						eGotoOpsStep	:= MagConvULStepSafetyBarRet;

						bPaused	:= p_bStop OR p_bStep;
					END_IF

				MagConvULStepMagCmp:
					sStepTxt	:= 'Comparing Magazine';

					a_tyMagAllwBffrStat[1]	:= p_tyBufferStat1;
					a_tyMagAllwBffrStat[2]	:= p_tyBufferStat2;
					a_tyMagAllwBffrStat[3]	:= p_tyBufferStat3;

					a_bMagAllwMagClamped[1]	:= p_bMagClampRS1;
					a_bMagAllwMagClamped[2]	:= p_bMagClampRS2;
					a_bMagAllwMagClamped[3]	:= p_bMagClampRS3;

					a_bMagAllwMagPresent[1]	:= p_bBufferMagPresent1 AND NOT(bMagExitedWait);
					a_bMagAllwMagPresent[2]	:= p_bBufferMagPresent2 AND NOT(p_bOpsMagConvUL2MagExitedWait);
					a_bMagAllwMagPresent[3]	:= p_bBufferMagPresent3 AND NOT(p_bOpsMagConvUL3MagExitedWait);

					IF NOT(bAutoRcpEn AND p_bMcParamMESEn) THEN
						a_udiMagAllwMagPresentTm[1]	:= DT_TO_UDINT(p_dtBufferMagPresentTm1);
						a_udiMagAllwMagPresentTm[2]	:= DT_TO_UDINT(p_dtBufferMagPresentTm2);
						a_udiMagAllwMagPresentTm[3]	:= DT_TO_UDINT(p_dtBufferMagPresentTm3);
					ELSE
						a_udiMagAllwMagPresentTm[1]	:= DT_TO_UDINT(p_dtOpsMagConvUL1AcptTm);
						a_udiMagAllwMagPresentTm[2]	:= DT_TO_UDINT(p_dtOpsMagConvUL2AcptTm);
						a_udiMagAllwMagPresentTm[3]	:= DT_TO_UDINT(p_dtOpsMagConvUL3AcptTm);

						a_iMagMESAcptCond[1] := p_iOpsMagConvUL1MESAcptCond;
						a_iMagMESAcptCond[2] := p_iOpsMagConvUL2MESAcptCond;
						a_iMagMESAcptCond[3] := p_iOpsMagConvUL3MESAcptCond;
					END_IF

					//Sorting Priority
					memset(ADR(a_udiMagAllwPriority), 0, SIZEOF(a_udiMagAllwPriority));

					FOR udi := 1 TO 3 DO
						udiCount	:= 3;
						udiCmpTm	:= a_udiMagAllwMagPresentTm[udi];

						FOR udi1 := 1 TO 3 DO
							IF a_udiMagAllwMagPresentTm[udi1] < udiCmpTm THEN
								udiCount	:= udiCount - 1;
							END_IF
						END_FOR

						a_udiMagAllwPriority[udi]	:= udiCount;
					END_FOR

//					FOR udi := 3 TO 1 BY -1 DO
//						FOR udi1 := 3 TO 1 BY -1 DO
//							IF (udi <> udi1) AND (a_udiMagAllwPriority[udi] = a_udiMagAllwPriority[udi1]) THEN
//								a_udiMagAllwPriority[udi1]	:= a_udiMagAllwPriority[udi1] - 1;
//							END_IF
//						END_FOR
//					END_FOR

					//Checking Buffer Status
					memset(ADR(a_udiMagAllwSum), 0, SIZEOF(a_udiMagAllwSum));

					FOR udi := 1 TO 3 DO
						//Priority
						a_udiMagAllwSum[udi]	:= a_udiMagAllwSum[udi] + a_udiMagAllwPriority[udi];
						//Enable
						IF pa_bMagDis[udi] = FALSE THEN
							a_udiMagAllwSum[udi]	:= a_udiMagAllwSum[udi] + 1000;
						END_IF
						//Magazine Clamped
						IF a_bMagAllwMagClamped[udi] = TRUE THEN
							a_udiMagAllwSum[udi]	:= a_udiMagAllwSum[udi] + 1000;
						END_IF
						//Magazine Present
						IF a_bMagAllwMagPresent[udi] = TRUE THEN
							a_udiMagAllwSum[udi]	:= a_udiMagAllwSum[udi] + 1000;
						END_IF
						//Magazine Empty
						IF a_tyMagAllwBffrStat[udi].bBffrMty = TRUE THEN
							a_udiMagAllwSum[udi]	:= a_udiMagAllwSum[udi] + 2500;
						END_IF
						//Magazine Available
						IF a_tyMagAllwBffrStat[udi].bBffrFull = FALSE AND a_tyMagAllwBffrStat[udi].bBffrMty = FALSE THEN
							a_udiMagAllwSum[udi]	:= a_udiMagAllwSum[udi] + 3000;
						END_IF
						//Magazine Reject
						IF pa_bMagRej[udi] = TRUE THEN
							a_udiMagAllwSum[udi]	:= a_udiMagAllwSum[udi] + 6000;
						END_IF
						//Customized Width Change
						IF bAutoRcpEn THEN
							IF pa_bMagChangeOverBlk[udi] = TRUE THEN
								a_udiMagAllwSum[udi]	:= a_udiMagAllwSum[udi] - 1000;
							END_IF
							IF p_bMcParamMESEn THEN
								IF a_iMagMESAcptCond[udi] = 0 AND  a_bMagAllwMagPresent [udi] THEN
									a_udiMagAllwSum[udi]	:= a_udiMagAllwSum[udi] - 1000;
								END_IF
							END_IF
						END_IF
					END_FOR

					udiMagAllwGo	:= 99;

					FOR udi := 1 TO 3 DO
						IF (a_udiMagAllwSum[udi] >= 6000 AND a_udiMagAllwSum[udi] < 7000 AND pa_bMagRej[usiMagConv] = FALSE)	//Enable + Magazine Clamped + Magazine Present + Magazine Available
							OR (a_udiMagAllwSum[udi] >= 12000 AND pa_bMagRej[usiMagConv] = TRUE) THEN							//Reject + Enable + Magazine Clamped + Magazine Present + Magazine Available

							IF udiMagAllwGo <> 99 THEN
								//Priority
								IF a_udiMagAllwSum[udi] > a_udiMagAllwSum[udiMagAllwGo] THEN
									udiMagAllwGo	:= udi;
								END_IF
							ELSE
								udiMagAllwGo	:= udi;
							END_IF

						END_IF

					END_FOR

					IF udiMagAllwGo = 99 THEN

						FOR udi := 1 TO 3 DO
							IF (a_udiMagAllwSum[udi] >= 5500 AND a_udiMagAllwSum[udi] < 7000 AND pa_bMagRej[usiMagConv] = FALSE)	//Enable + Magazine Clamped + Magazine Present + Magazine Empty
								OR (a_udiMagAllwSum[udi] >= 11500 AND pa_bMagRej[usiMagConv] = TRUE) THEN							//Reject + Enable + Magazine Clamped + Magazine Present + Magazine Empty

								IF udiMagAllwGo <> 99 THEN
									//Priority
									IF a_udiMagAllwSum[udi] > a_udiMagAllwSum[udiMagAllwGo] THEN
										udiMagAllwGo	:= udi;
									END_IF
								ELSE
									udiMagAllwGo	:= udi;
								END_IF

							END_IF

						END_FOR

					END_IF

					IF p_bRlsMag = TRUE THEN
						eGotoOpsStep	:=MagConvULStepMagExitMnl;
					ELSIF (p_bDISOTAGVReady OR
						  pa_bMagChangeOverBlk[p_usiMagConv] )
						AND (p_eCustomerReq = Siemens OR p_eCustomerReq = We_Fabricate )THEN
						eGotoOpsStep	:= MagConvULStepMagExitClampCtrl;
					ELSIF p_tyLocalBufferStat.bBffrFull = TRUE AND p_bOutShutterExtended OR (p_bUSAllow = FALSE AND NOT(bAutoRcpEn)) THEN
					//	eGotoOpsStep    := MagConvULStepMagFullDSComm;
						eGotoOpsStep	:= MagConvULStepMagExitClampCtrl;
					ELSIF NOT(p_bUSAllow) AND bAutoRcpEn AND  udiMagAllwGo = p_usiMagConv THEN
						//do nothing when blocking
						sStepTxt	:= 'Comparing Mag: Waiting available magazine to change width';
						bPaused	:= p_bStop;
					ELSIF p_bAllwChgWidth AND bAutoRcpEn THEN
						eGotoOpsStep	:= 	MagConvULStepMagAWEngage;
					ELSIF p_bAllwChgSlot AND bAutoRcpEn THEN
						eGotoOpsStep := MagConvULStepMtyBffr;
					ELSE

						IF (p_bUSAllow = TRUE) AND (udiMagAllwGo <> 99) THEN

							IF udiMagAllwGo = p_usiMagConv THEN
								bMagBffrAvl		:= TRUE;
//								IF NOT(bAutoRcpEn AND p_tyLocalBufferStat.bBffrMty = TRUE) THEN
									eGotoOpsStep	:= MagConvULStepNxtLoadBffr;
//								ELSE
//									eGotoOpsStep	:= MagConvULStepMtyBffr;
//								END_IF

								bPaused	:= p_bStop OR p_bStep;
							ELSE
								bPaused	:= p_bStop;
							END_IF

						ELSE
							bPaused	:= p_bStop;
						END_IF

					END_IF
				MagConvULStepMtyBffr:
					sStepTxt	:= 'Resetting Buffer Setting';
					eBufferAct := BufferActSetMty;

					IF p_eBufferStatus = Done AND p_eBufferStat = BufferActSetMty THEN
						eBufferAct		:= BufferActIdle;
						eGotoOpsStep	:= MagConvULStepMagCmp;

						bPaused	:= p_bStop OR p_bStep;
					END_IF

				MagConvULStepNxtLoadBffr:
					sStepTxt	:= 'Computing Next Load Buffer';

					eBufferAct	:= BufferActNxtLoad;

					IF p_eBufferStatus = Done AND p_eBufferStat = BufferActNxtLoad THEN
						eBufferAct		:= BufferActIdle;
						eGotoOpsStep	:= MagConvULStepBffrUSComm;

						bPaused	:= p_bStop OR p_bStep;
					END_IF

				MagConvULStepBffrUSComm:
					sStepTxt	:= 'Communicating Buffer Upstream';

					eUSSMEMAAct	:= SMEMAActRun;

					IF p_bUSSMEMATransporting = TRUE THEN
						eGotoOpsStep	:= MagConvULStepBffrEntBrd;
						IF p_eNtParamProjMagBuffferActLoad = BufferActLoadWhenStarted
							THEN

							eBufferAct	:= BufferActLoad;
						END_IF
					ELSIF p_bRlsMag = TRUE AND (p_bOpsTravLifAllwExitMag OR p_eCustomerReq <> Siemens) THEN
						bMagBffrAvl		:= FALSE;
						eUSSMEMAAct		:= SMEMAActIdle;
						eGotoOpsStep	:= MagConvULStepMagExitMnl;

					ELSIF  ((p_bAllwChgWidth OR p_bAllwChgSlot) AND NOT(p_bMcParamAutoRcpDis) )  OR p_bUSAllow = FALSE  THEN//IF needed to insert back to Previous Magazine
						bMagBffrAvl		:= FALSE;
						eUSSMEMAAct		:= SMEMAActIdle;
						eGotoOpsStep	:= MagConvULStepMagCmp;

						bPaused	:= p_bStop OR p_bStep;

					ELSIF (p_tyLocalBufferStat.bBffrFull = TRUE ) //AND p_bOutShutterExtended OR p_eCustomerReq = Siemens
						OR (p_bDISOTAGVReady AND p_bOpsTravLifAllwExitMag) THEN //OR  p_bUSAllow = FALSE THEN
						bMagBffrAvl		:= FALSE;
						eUSSMEMAAct		:= SMEMAActIdle;
					//	eGotoOpsStep    := MagConvULStepMagFullDSComm;
						eGotoOpsStep    := MagConvULStepMagExitClampCtrl;
					ELSE

						IF pa_bMagDis[usiMagConv] = TRUE THEN		//Checking Magazine Enable
							bMagBffrAvl		:= FALSE;
							eGotoOpsStep	:= MagConvULStepMagCmp;

							bPaused	:= p_bStop OR p_bStep;
						ELSE
							bPaused	:= p_bStop;
						END_IF

						IF bPaused = TRUE OR pa_bMagDis[usiMagConv] = TRUE THEN
							eUSSMEMAAct	:= SMEMAActIdle;
						END_IF

					END_IF

				MagConvULStepBffrEntBrd:
					IF p_bUSSMEMATransporting AND EDGEPOS(p_bUSSMEMAConvStart) THEN
						sStepTxt	:= 'Transferring Board Into Magazine';
						IF p_eNtParamProjMagBuffferActLoad = BufferActLoadWhenStarted
							THEN

							eBufferAct	:= BufferActLoad;
						END_IF

					END_IF

					IF p_bUSSMEMATransporting AND EDGEPOS(p_bUSSMEMAConvStop) THEN
						sStepTxt	:= 'Stop Transferring';
						//Do Nothing
					END_IF

//					IF p_bUSSMEMATransporting = FALSE
//						THEN
//						eGotoOpsStep	:= MagConvULStepBffrUSComm;
//					END_IF

					IF (p_eUSSMEMAStatus = Done AND p_eUSSMEMAStat = SMEMAActRun)
						AND (p_eConvStat = ConvActExitPshr AND p_eConvStatus = Done)
						THEN
						eUSSMEMAAct		:= SMEMAActIdle;
						eGotoOpsStep	:= MagConvULStepLoadBffr;
					END_IF

				MagConvULStepLoadBffr:
					sStepTxt	:= 'Loading Buffer';

					eBufferAct	:= BufferActLoad;

					IF p_eBufferStatus = Done AND p_eBufferStat = BufferActLoad THEN
						eBufferAct		:= BufferActIdle;
						bMagBffrAvl		:= FALSE;
						eGotoOpsStep	:= MagConvULStepBffrStatChk;

						bPaused	:= p_bStop OR p_bStep;
					END_IF
				MagConvULStepMagExtMESStdByChk:
					sStepTxt	:= 'Mag StdBy for MES response Before Exiting';
					bWriteRFID := TRUE;
					fbWriteRFIDTO(IN:= bWriteRFID,PT := DINT_TO_TIME(p_diMcParamMESResponseTO) );
					IF p_tyResponseFromMES.bRFIDWriteComplete  THEN //Accept
						IF ePrevStepBeforeMESStdBy = MagConvULStepMagExitMnl THEN
							eGotoOpsStep := MagConvULStepMagExitMnl;
						ELSIF ePrevStepBeforeMESStdBy = MagConvULStepMagExitClampCtrl THEN
							eGotoOpsStep := MagConvULStepMagExitClampCtrl;
						END_IF
					ELSIF fbWriteRFIDTO.Q  AND p_bRlsMag THEN
						sStepTxt	:= 'MES response to Write RFID Timeout, Press Rls Mag to Manual Exit ';

						eGotoOpsStep := MagConvULStepMagExitMnl;

					END_IF

					bPaused	:= p_bStop OR p_bStep;

				MagConvULStepMagExitClampCtrl:
					sStepTxt	:= 'Extending Selection Clamp';

					eSelClampCtrl := PneuActExt;
					eMagAWEngageAct	:= PneuActRet;
					ePrevExitStep := MagConvULStepMagExitClampCtrl;
					IF (p_eSelClampCtrlStat = PneuActExt AND p_eSelClampCtrlStatus = Done)
						OR (p_eMagAWEngageStat = PneuActRet AND p_eMagAWEngageStatus = Done)
						THEN
						eMagAWEngageAct	:= PneuActIdle;
						eSelClampCtrl	:= PneuActIdle;
						eGotoOpsStep    := MagConvULStepMagExitSafeBarCtrl;
						bPaused	:= p_bStop OR p_bStep;
					END_IF

				MagConvULStepMagExitSafeBarCtrl:
					IF p_bSafetyBarExtended = FALSE THEN
						eSafetyBarAct	:= PneuActExt;

						IF p_eSafetyBarStatus = Done AND p_eSafetyBarStat = PneuActExt THEN
							eSafetyBarAct	:= PneuActIdle;
							eGotoOpsStep    := MagConvULStepMagFullDSComm;

							bPaused	:= p_bStop OR p_bStep;
						END_IF
					ELSE
						eGotoOpsStep    := MagConvULStepMagFullDSComm;
					END_IF

				MagConvULStepMagFullDSComm:
					sStepTxt	:= 'Communicating AGV Machine And Ready Exit';

					eAGVMagAct	:= AGVMagActExit;
					IF bMagAutoEx THEN
						eDSSOTAct	:= SOTActRun;
					ELSE
						eDSSOTAct	:= SOTActIdle;
					END_IF

					IF p_bAGVMagMcRunRdy = TRUE THEN
						eGotoOpsStep	:= MagConvULStepMagFullExit;

					ELSIF p_bRlsMag = TRUE
						OR (p_tyLocalBufferStat.bBffrFull AND p_bDIOutShutterClosedRS ) //AND p_bOutShutterExtended )
						OR (pa_bMagChangeOverBlk[p_usiMagConv] = TRUE AND bAutoRcpEn)
						OR (p_bUSAllow = FALSE AND NOT(bAutoRcpEn) )THEN
						eAGVMagAct		:= AGVMagActIdle;
						eGotoOpsStep	:= MagConvULStepMagExitMnl;

					ELSE
						bPaused	:= p_bStop;

						IF bPaused = TRUE THEN
							eAGVMagAct	:= AGVMagActIdle;
						END_IF

					END_IF

				MagConvULStepMagFullExit:
					sStepTxt	:= 'Magazine Conveyor Exiting Magazine';

					eMagConv2ClpAct	:= MagConv2ClpActExitClpr;
					eSelClampCtrl	:= PneuActExt;

					IF ((p_eAGVMagStatus = Done AND p_eAGVMagStat = AGVMagActExit)
						OR (p_eDSSOTStatus = Done AND p_eDSSOTStat = SOTActRun))
						AND (p_eMagConv2ClpStatus = Done AND p_eMagConv2ClpStat = MagConv2ClpActExitClpr)
						AND (p_eSelClampCtrlStatus = Done AND p_eSelClampCtrlStat = PneuActExt)
						THEN
						eDSSOTAct			:= SOTActIdle;
						eAGVMagAct			:= AGVMagActIdle;
						eMagConv2ClpAct		:= MagConv2ClpActIdle;
						eSelClampCtrl		:= PneuActIdle;
						eGotoOpsStep		:= MagConvULStepMagExitedAGVWait;
						bMagSizeLarge := FALSE;
						bPaused	:= p_bStop OR p_bStep;
					END_IF

				MagConvULStepMagExitedAGVWait:
					sStepTxt  := 'Magazine Exited and wait for AGV Leave';

					IF bAIVInPos = FALSE OR p_bBufferMagRemoved THEN
						ePrevExitStep 		:= MagConvULStepNA;
						iMagMESAcptCond 	:= 0;
						eGotoOpsStep        := MagConvULStepMagUSComm;
						eDSSOTAct			:= SOTActIdle;

					END_IF

					bPaused   := p_bStop OR p_bStep;

				MagConvULStepMagExitMnl:
					sStepTxt	:= 'Magazine Conveyor Exiting Magazine Manually';
					IF p_bProjLifTravMnlLoad = FALSE THEN
						eMagConv2ClpAct	:= MagConv2ClpActPreExitClpr;
						eSelClampCtrl	:= PneuActExt;
						eSafetyBarAct	:= PneuActExt;
					ELSE
						eGotoOpsStep		:= MagConvULStepMagExitedWait; //no roller
					END_IF
					ePrevExitStep := MagConvULStepMagExitMnl;
					IF ((p_eMagConv2ClpStatus = Done AND p_eMagConv2ClpStat = MagConv2ClpActPreExitClpr)  OR EDGENEG(p_bDIMagFixedClampSen))
						AND (p_eSelClampCtrlStatus = Done AND p_eSelClampCtrlStat = PneuActExt)
						AND (p_eSafetyBarStatus = Done AND p_eSafetyBarStat = PneuActExt)
						THEN
						eSelClampCtrl	:= PneuActIdle;
						eSafetyBarAct	:= PneuActIdle;
						eMagConv2ClpAct		:= MagConv2ClpActIdle;
						eGotoOpsStep		:= MagConvULStepMagExitedWait;

						bPaused	:= p_bStop OR p_bStep;
					END_IF

				MagConvULStepMagExitedWait:
					sStepTxt	:= 'Magazine Exited And Waiting For Remove';
					eAGVMagAct 	:= AGVMagActExit;
					IF bMagAutoEx THEN
						eDSSOTAct			:= SOTActRun;
					ELSE
						eDSSOTAct			:= SOTActIdle;
					END_IF

					bMagExitedWait	:= TRUE;

					fbEntSenOff(IN:= p_bLocalMagEntrySen = FALSE AND (NOT((p_bLocalBufferMagPresent OR p_bMag1OrientationChkSen1) AND p_bProjLifTravMnlLoad))); //p_bMag1OrientationChkSen1
					IF fbMagRemovedTm.Q OR fbEntSenOff.Q THEN
						bMagExitedWait	:= FALSE;
						ePrevExitStep 		:= MagConvULStepNA;
						iMagMESAcptCond 	:= 0;
						eGotoOpsStep	:= MagConvULStepMagUSComm;
						eDSSOTAct	:= SOTActIdle;

					ELSIF p_bNewMag = TRUE THEN
						bMagExitedWait	:= FALSE;
						eAGVMagAct 	:= AGVMagActIdle;
						ePrevExitStep 		:= MagConvULStepNA;
						iMagMESAcptCond 	:= 0;
						eGotoOpsStep	:= MagConvULStepMagEntMnl;
						eDSSOTAct			:= SOTActIdle;
					END_IF

					IF p_bAGVMagMcRunRdy = TRUE THEN
						eGotoOpsStep 	:= MagConvULStepMagFullExit;
					ELSIF p_bDSSOTConvStart= TRUE THEN
						eGotoOpsStep 	:= MagConvULStepMagFullExit;
					END_IF

					bPaused	:= p_bStop OR p_bStep;

			END_CASE

		END_IF

	END_IF

	bNewMagAllw	:= eOpsStep = MagConvULStepMagUSComm;

	bRlsMagAllw	:= ((eOpsStep = MagConvULStepMagCmp
					OR eOpsStep = MagConvULStepBffrUSComm
					OR eOpsStep = MagConvULStepMagFullDSComm
					OR eOpsStep = MagConvULStepBffrEntBrd
					OR (eOpsStep = MagConvULStepMagEntMESStdByChk AND fbReadRFIDTO.Q )
					OR (eOpsStep = MagConvULStepMagExtMESStdByChk AND fbWriteRFIDTO.Q) )
					);

	bEjectMESStep		:= 	eGotoOpsStep =  MagConvULStepMagExitMnl;//eOpsStep = MagConvULStepMagEntMESStdByChk OR eOpsStep = MagConvULStepMagExtMESStdByChk	;
	bEjectMagNotAllw	:= FALSE;//NOT((eOpsStep = MagConvULStepMagEntMESStdByChk AND fbReadRFIDTO.Q)
						//OR (eOpsStep = MagConvULStepMagExtMESStdByChk AND fbWriteRFIDTO.Q));

	Act_OpsInfo;

	//Operation State
	bOpsInitDone				:= eOpsStep > MagConvULStepInitMagConv;
	bStepMagExitedWait			:= eOpsStep = MagConvULStepMagExitedWait;
	bStepMagVerification 		:= eOpsStep = MagConvULStepVerifyMag;
	bStepMagFullExit 			:= eOpsStep = MagConvULStepMagFullExit;
	bStepMagUSCom 				:= eOpsStep = MagConvULStepMagUSComm;
	bStepMagBffrLoad		    := eOpsStep > MagConvULStepMagUSComm;
	bAGVComm1Rdy				:= (eOpsStep = MagConvULStepMagUSComm OR eOpsStep = MagConvULStepMagFullDSComm OR eOpsStep = MagConvULStepMagExitedWait
								    OR eOpsStep = MagConvULStepMagEnt OR eOpsStep = MagConvULStepMagFullExit) AND p_bAGVMagMcRunRdy;
	bStepOpsMagAWDone 			:= eOpsStep = MagConvULStepMagAWMov AND eGotoOpsStep = MagConvULStepMagAWDisengage;
	bStepOpsPitchUpdated		:= eOpsStep = MagConvULStepMtyBffr AND eGotoOpsStep = MagConvULStepMagCmp;
	bStepPLCGrab				:= p_tyLocalBufferStat.bBffrMty AND EDGEPOS(p_bMagPresentSen);

END_ACTION
```

### OpsMagConvUL2.var - Change By Project
```iecst
(*2019-03-25*)
(**)
(*Action & State & Status*)
(**)
(*Alarm*)
VAR
	p_OpsMagConvUL2AlmData : UDINT;
	p_OpsMagConvUL2AlmData1 : UDINT;
END_VAR
(**)
(*Output*)
VAR
	p_OpsMagConvUL2StepTxt : UDINT;
	p_OpsMagConvUL2Paused : UDINT;
END_VAR
(**)
VAR
	p_OpsMagConvUL2BufferAct : UDINT;
	p_OpsMagConvUL2MagConv2ClpAct : UDINT;
	p_OpsMagConvUL2USSMEMAAct : UDINT;
	p_OpsMagConvUL2AGVMagAct : UDINT;
	p_OpsMagConvUL2MagFullExit : UDINT;
	p_OpsMagConvUL2IncorrectMagModel : UDINT;
	p_OpsMagConvUL2MagSizeL : UDINT;
END_VAR
(**)
VAR
	p_OpsMagConvUL2InitDone : UDINT;
	p_OpsMagConvUL2MagBffrAvl : UDINT;
	p_OpsMagConvUL2NewMagAllw : UDINT;
	p_OpsMagConvUL2RlsMagAllw : UDINT;
	p_OpsMagConvUL2EjectMESStep : UDINT;
	p_OpsMagConvUL2EjectMagNotAllw : UDINT;
	p_OpsMagConvUL2StepSelClampCtrl : UDINT;
	p_OpsMagConvUL2StepMagExitedWait : UDINT;
	p_OpsMagConvUL2NewMagVerified : UDINT;
	p_OpsMagConvUL2StepUSCom : UDINT;
	p_OpsMagConvUL2StepPLCGrab : UDINT;
END_VAR
(**)
VAR
	p_OpsMagConvUL2SafetyBarAct : UDINT;
	p_OpsMagConvUL2MagAWEngageAct : UDINT;
	p_OpsMagConvUL2MagAWAct : UDINT;
	p_OpsAGVCommRdy2 : UDINT;
END_VAR
(**)
VAR
	p_OpsMagConvUL2USSOTAct : UDINT;
	p_OpsMagConvUL2DSSOTAct : UDINT;
	p_OpsMagConvUL2UnclmpDone : UDINT;
	p_OpsMagConvUL2MagAllwGo : UDINT;
	p_OpsMagConvUL2ReadRFID : UDINT;
	p_OpsMagConvUL2WriteRFID : UDINT;
	p_OpsMagConvUL2AWDone : UDINT;
	p_OpsMagConvUL2SlotUpdtDone : UDINT;
	p_OpsMagConvUL2AcptTm : UDINT;
	p_OpsMagConvUL2MESAcptCond : UDINT;
	p_OpsMagConvUL2MagExitedWait : UDINT;
END_VAR
```

### Program Logical/Operations/MagConv_StationaryPlat/OpsMagConvUL2 (IEC, version 1.00.0) - 1.00.0 - 

#### Init.st - Change By Project
```iecst
(** 2019-03-25 **)
PROGRAM _INIT

	(* Always Change If Project Change *)

	//Physical Configuration
	usiMagConv	:= 2;

	//Pass Address To Global Address For External Use
	//Action, State & Status

	//Alarm
	p_OpsMagConvUL2AlmData	:= ADR(tyAlmData);
	p_OpsMagConvUL2AlmData1	:= ADR(tyAlmData1);

	//Output
	p_OpsMagConvUL2StepTxt	:= ADR(sStepTxt);
	p_OpsMagConvUL2Paused	:= ADR(bPaused);

	p_OpsMagConvUL2BufferAct		:= ADR(eBufferAct);
	p_OpsMagConvUL2MagConv2ClpAct	:= ADR(eMagConv2ClpAct);
	p_OpsMagConvUL2USSMEMAAct		:= ADR(eUSSMEMAAct);
	p_OpsMagConvUL2AGVMagAct		:= ADR(eAGVMagAct);

	p_OpsMagConvUL2InitDone				:= ADR(bOpsInitDone);
	p_OpsMagConvUL2MagBffrAvl			:= ADR(bMagBffrAvl);
	p_OpsMagConvUL2NewMagAllw			:= ADR(bNewMagAllw);
	p_OpsMagConvUL2RlsMagAllw			:= ADR(bRlsMagAllw);
	p_OpsMagConvUL2EjectMESStep			:= ADR(bEjectMESStep); //MES
	p_OpsMagConvUL2EjectMagNotAllw		:= ADR(bEjectMagNotAllw); //MES
	p_OpsMagConvUL2StepMagExitedWait	:= ADR(bStepMagExitedWait);
	p_OpsMagConvUL2StepUSCom			:= ADR(bStepMagUSCom);
	p_OpsMagConvUL2StepPLCGrab			:= ADR(bStepPLCGrab);

	p_OpsMagConvUL2StepSelClampCtrl		:= ADR(eSelClampCtrl);
	p_OpsMagConvUL2NewMagVerified		:= ADR(bNewMagVerified);
	p_OpsMagConvUL2MagFullExit			:= ADR(bStepMagFullExit);
	p_OpsMagConvUL2IncorrectMagModel    := ADR(bIncorrectMagazineModel);
	p_OpsMagConvUL2MagSizeL    			:= ADR(bMagSizeLarge);

	p_OpsMagConvUL2SafetyBarAct			:= ADR(eSafetyBarAct);
	p_OpsMagConvUL2MagAWEngageAct		:= ADR(eMagAWEngageAct);
	p_OpsMagConvUL2MagAWAct				:= ADR(eMagAWAct);

	p_OpsMagConvUL2USSOTAct				:= ADR(eUSSOTAct);
	p_OpsMagConvUL2DSSOTAct				:= ADR(eDSSOTAct);

	p_OpsAGVCommRdy2					:= ADR(bAGVComm2Rdy);

	p_OpsMagConvUL2UnclmpDone			:= ADR(bPneuUnclmpDone);
	p_OpsMagConvUL2MagAllwGo			:= ADR(udiMagAllwGo);

	p_OpsMagConvUL2ReadRFID				:= ADR(bReadRFID);
	p_OpsMagConvUL2WriteRFID			:= ADR(bWriteRFID);
	p_OpsMagConvUL2AWDone			 	:= ADR(bStepOpsMagAWDone);
	p_OpsMagConvUL2SlotUpdtDone			:= ADR(bStepOpsPitchUpdated);
	(* Always Change If Project Change *)

	p_OpsMagConvUL2AcptTm				:= ADR(dtMagConvAcptTm);
	p_OpsMagConvUL2MESAcptCond 			:= ADR(iMagMESAcptCond);
	p_OpsMagConvUL2MagExitedWait 		:= ADR(bMagExitedWait);
END_PROGRAM
```
